LIN {X 0,Y 132.455,Z 460.625,A -85,B 0,C 180,E1 -25055.709,E2 -25055.709} C_VEL
LIN {X 0,Y 133.664,Z 463.302,A -85,B 0,C 180,E1 -25057.206,E2 -25057.206} C_VEL
LIN {X 0,Y 135.745,Z 466.18,A -85,B 0,C 180,E1 -25059.267,E2 -25059.267} C_VEL
LIN {X 0,Y 139.703,Z 473.299,A -85,B 0,C 180,E1 -25063.516,E2 -25063.516} C_VEL
LIN {X 0,Y 143.057,Z 480.754,A -85,B 0,C 180,E1 -25067.47,E2 -25067.47} C_VEL
LIN {X 0,Y 145.337,Z 487.251,A -85,B 0,C 180,E1 -25070.689,E2 -25070.689} C_VEL
LIN {X 0,Y 147.51,Z 495.449,A -85,B 0,C 180,E1 -25074.692,E2 -25074.692} C_VEL
LIN {X 0,Y 148.704,Z 503.562,A -85,B 0,C 180,E1 -25078.676,E2 -25078.676} C_VEL
LIN {X 0,Y 148.492,Z 505.004,A -85,B 0,C 180,E1 -25079.314,E2 -25079.314} C_VEL
LIN {X 0,Y 144.709,Z 513.242,A -85,B 0,C 180,E1 -25082.524,E2 -25082.524} C_VEL
LIN {X 0,Y 140.761,Z 521.094,A -85,B 0,C 180,E1 -25086.458,E2 -25086.458} C_VEL
LIN {X 0,Y 137.597,Z 527.354,A -85,B 0,C 180,E1 -25090.61,E2 -25090.61} C_VEL
LIN {X 0,Y 134.854,Z 532.346,A -85,B 0,C 180,E1 -25094.896,E2 -25094.896} C_VEL
LIN {X 0,Y 132.714,Z 536.229,A -85,B 0,C 180,E1 -25099.319,E2 -25099.319} C_VEL
LIN {X 0,Y 131.093,Z 539.121,A -85,B 0,C 180,E1 -25103.845,E2 -25103.845} C_VEL
LIN {X 0,Y 130.431,Z 540.5,A -85,B 0,C 180,E1 -25106.912,E2 -25106.912} C_VEL
LIN {X 0,Y 130.214,Z 542.071,A -85,B 0,C 180,E1 -25113.095,E2 -25113.095} C_VEL
LIN {X 0,Y 130.346,Z 542.325,A -85,B 0,C 180,E1 -25116.191,E2 -25116.191} C_VEL
LIN {X 0,Y 130.708,Z 542.169,A -85,B 0,C 180,E1 -25119.283,E2 -25119.283} C_VEL
LIN {X 0,Y 133.029,Z 540.615,A -85,B 0,C 180,E1 -25125.317,E2 -25125.317} C_VEL
LIN {X 0,Y 134.623,Z 539.262,A -85,B 0,C 180,E1 -25128.255,E2 -25128.255} C_VEL
LIN {X 0,Y 137.536,Z 536.056,A -85,B 0,C 180,E1 -25133.103,E2 -25133.103} C_VEL
LIN {X 0,Y 141.54,Z 531.107,A -85,B 0,C 180,E1 -25138.146,E2 -25138.146} C_VEL
LIN {X 0,Y 145.353,Z 525.767,A -85,B 0,C 180,E1 -25142.132,E2 -25142.132} C_VEL
LIN {X 0,Y 149.813,Z 519.05,A -85,B 0,C 180,E1 -25145.903,E2 -25145.903} C_VEL
LIN {X 0,Y 152.887,Z 513.993,A -85,B 0,C 180,E1 -25148.135,E2 -25148.135} C_VEL
LIN {X 0,Y 153.42,Z 512.528,A -85,B 0,C 180,E1 -25148.853,E2 -25148.853} C_VEL
LIN {X 0,Y 153.039,Z 506.128,A -85,B 0,C 180,E1 -25152.712,E2 -25152.712} C_VEL
LIN {X 0,Y 152.175,Z 500.29,A -85,B 0,C 180,E1 -25156.151,E2 -25156.151} C_VEL
LIN {X 0,Y 150.593,Z 493.774,A -85,B 0,C 180,E1 -25160.084,E2 -25160.084} C_VEL
LIN {X 0,Y 148.374,Z 487.095,A -85,B 0,C 180,E1 -25164.311,E2 -25164.311} C_VEL
LIN {X 0,Y 146.121,Z 481.755,A -85,B 0,C 180,E1 -25168.057,E2 -25168.057} C_VEL
LIN {X 0,Y 143.486,Z 476.383,A -85,B 0,C 180,E1 -25172.267,E2 -25172.267} C_VEL
LIN {X 0,Y 141.705,Z 473.457,A -85,B 0,C 180,E1 -25175.066,E2 -25175.066} C_VEL
LIN {X 0,Y 140.997,Z 471.644,A -85,B 0,C 180,E1 -25176.499,E2 -25176.499} C_VEL
LIN {X 0,Y 140.073,Z 470.683,A -85,B 0,C 180,E1 -25177.895,E2 -25177.895} C_VEL
LIN {X 0,Y 138.51,Z 471.715,A -85,B 0,C 180,E1 -25179.195,E2 -25179.195} C_VEL
LIN {X 0,Y 137.186,Z 472.293,A -85,B 0,C 180,E1 -25180.549,E2 -25180.549} C_VEL
LIN {X 0,Y 136.277,Z 473.332,A -85,B 0,C 180,E1 -25181.196,E2 -25181.196} C_VEL
LIN {X 0,Y 134.058,Z 476.489,A -85,B 0,C 180,E1 -25182.544,E2 -25182.544} C_VEL
LIN {X 0,Y 133.026,Z 477.829,A -85,B 0,C 180,E1 -25183.286,E2 -25183.286} C_VEL
LIN {X 0,Y 131.762,Z 479.038,A -85,B 0,C 180,E1 -25184.532,E2 -25184.532} C_VEL
LIN {X 0,Y 131.276,Z 479.221,A -85,B 0,C 180,E1 -25185.294,E2 -25185.294} C_VEL
LIN {X 0,Y 131.17,Z 478.619,A -85,B 0,C 180,E1 -25186.101,E2 -25186.101} C_VEL
LIN {X 0,Y 130.057,Z 490.324,A -85,B 0,C 180,E1 -25189.885,E2 -25189.885} C_VEL
LIN {X 0,Y 129.323,Z 500.383,A -85,B 0,C 180,E1 -25193.76,E2 -25193.76} C_VEL
LIN {X 0,Y 129.054,Z 510.666,A -85,B 0,C 180,E1 -25198.439,E2 -25198.439} C_VEL
LIN {X 0,Y 129.652,Z 520.617,A -85,B 0,C 180,E1 -25203.885,E2 -25203.885} C_VEL
LIN {X 0,Y 131.03,Z 528.937,A -85,B 0,C 180,E1 -25209.259,E2 -25209.259} C_VEL
LIN {X 0,Y 134.097,Z 536.791,A -85,B 0,C 180,E1 -25215.191,E2 -25215.191} C_VEL
LIN {X 0,Y 138.864,Z 543.178,A -85,B 0,C 180,E1 -25220.749,E2 -25220.749} C_VEL
LIN {X 0,Y 144.895,Z 548.225,A -85,B 0,C 180,E1 -25225.883,E2 -25225.883} C_VEL
LIN {X 0,Y 152.196,Z 551.996,A -85,B 0,C 180,E1 -25230.527,E2 -25230.527} C_VEL
LIN {X 0,Y 160.602,Z 554.573,A -85,B 0,C 180,E1 -25234.672,E2 -25234.672} C_VEL
LIN {X 0,Y 171.114,Z 556.077,A -85,B 0,C 180,E1 -25238.705,E2 -25238.705} C_VEL
LIN {X 0,Y 173.413,Z 556.275,A -85,B 0,C 180,E1 -25239.643,E2 -25239.643} C_VEL
LIN {X 0,Y 164.631,Z 559.404,A -85,B 0,C 180,E1 -25243.47,E2 -25243.47} C_VEL
LIN {X 0,Y 151.897,Z 562.596,A -85,B 0,C 180,E1 -25249.626,E2 -25249.626} C_VEL
LIN {X 0,Y 144.624,Z 563.745,A -85,B 0,C 180,E1 -25254.327,E2 -25254.327} C_VEL
LIN {X 0,Y 137.24,Z 563.903,A -85,B 0,C 180,E1 -25260.982,E2 -25260.982} C_VEL
LIN {X 0,Y 136.599,Z 564.145,A -85,B 0,C 180,E1 -25261.627,E2 -25261.627} C_VEL
LIN {X 0,Y 132.236,Z 569.84,A -85,B 0,C 180,E1 -25266.508,E2 -25266.508} C_VEL
LIN {X 0,Y 129.732,Z 573.62,A -85,B 0,C 180,E1 -25271.031,E2 -25271.031} C_VEL
LIN {X 0,Y 128.674,Z 575.62,A -85,B 0,C 180,E1 -25274.151,E2 -25274.151} C_VEL
LIN {X 0,Y 127.892,Z 578.343,A -85,B 0,C 180,E1 -25280.51,E2 -25280.51} C_VEL
LIN {X 0,Y 128.152,Z 579.135,A -85,B 0,C 180,E1 -25283.702,E2 -25283.702} C_VEL
LIN {X 0,Y 128.639,Z 579.512,A -85,B 0,C 180,E1 -25286.867,E2 -25286.867} C_VEL
LIN {X 0,Y 129.364,Z 579.441,A -85,B 0,C 180,E1 -25289.999,E2 -25289.999} C_VEL
LIN {X 0,Y 128.652,Z 578.72,A -85,B 0,C 180,E1 -25293.131,E2 -25293.131} C_VEL
LIN {X 0,Y 127.97,Z 576.442,A -85,B 0,C 180,E1 -25298.683,E2 -25298.683} C_VEL
LIN {X 0,Y 128.234,Z 572.826,A -85,B 0,C 180,E1 -25304.277,E2 -25304.277} C_VEL
LIN {X 0,Y 129.379,Z 568.573,A -85,B 0,C 180,E1 -25309.021,E2 -25309.021} C_VEL
LIN {X 0,Y 132.123,Z 562.165,A -85,B 0,C 180,E1 -25314.345,E2 -25314.345} C_VEL
LIN {X 0,Y 134.691,Z 556.486,A -85,B 0,C 180,E1 -25318.008,E2 -25318.008} C_VEL
LIN {X 0,Y 137.421,Z 547.961,A -85,B 0,C 180,E1 -25322.478,E2 -25322.478} C_VEL
LIN {X 0,Y 140.149,Z 538.592,A -85,B 0,C 180,E1 -25326.413,E2 -25326.413} C_VEL
LIN {X 0,Y 142.414,Z 528.505,A -85,B 0,C 180,E1 -25329.906,E2 -25329.906} C_VEL
LIN {X 0,Y 144.054,Z 517.734,A -85,B 0,C 180,E1 -25333.079,E2 -25333.079} C_VEL
LIN {X 0,Y 145.067,Z 506.101,A -85,B 0,C 180,E1 -25336.048,E2 -25336.048} C_VEL
LIN {X 0,Y 145.054,Z 495.817,A -85,B 0,C 180,E1 -25338.484,E2 -25338.484} C_VEL
LIN {X 0,Y 142.546,Z 488.232,A -85,B 0,C 180,E1 -25341.052,E2 -25341.052} C_VEL
LIN {X 0,Y 139.792,Z 481.393,A -85,B 0,C 180,E1 -25343.582,E2 -25343.582} C_VEL
LIN {X 0,Y 137.388,Z 475.79,A -85,B 0,C 180,E1 -25345.758,E2 -25345.758} C_VEL
LIN {X 0,Y 135.102,Z 471.173,A -85,B 0,C 180,E1 -25347.778,E2 -25347.778} C_VEL
LIN {X 0,Y 134.46,Z 469.699,A -85,B 0,C 180,E1 -25348.378,E2 -25348.378} C_VEL
LIN {X 0,Y 131.756,Z 465.595,A -85,B 0,C 180,E1 -25350.738,E2 -25350.738} C_VEL
LIN {X 0,Y 130.923,Z 463.575,A -85,B 0,C 180,E1 -25351.576,E2 -25351.576} C_VEL
LIN {X 0,Y 130.035,Z 462.484,A -85,B 0,C 180,E1 -25352.488,E2 -25352.488} C_VEL
LIN {X 0,Y 123.354,Z 459.002,A -85,B 0,C 180,E1 -25361.308,E2 -25361.308} C_VEL
LIN {X 0,Y 122.315,Z 457.065,A -85,B 0,C 180,E1 -25365.126,E2 -25365.126} C_VEL
LIN {X 0,Y 122.285,Z 456.255,A -85,B 0,C 180,E1 -25367.175,E2 -25367.175} C_VEL
LIN {X 0,Y 122.406,Z 456.239,A -85,B 0,C 180,E1 -25370.082,E2 -25370.082} C_VEL
LIN {X 0,Y 122.6,Z 456.214,A -85,B 0,C 180,E1 -25376.714,E2 -25376.714} C_VEL
LIN {X 0,Y 123.044,Z 456.158,A -85,B 0,C 180,E1 -25380.001,E2 -25380.001} C_VEL
LIN {X 0,Y 122.422,Z 456.217,A -85,B 0,C 180,E1 -25387.189,E2 -25387.189} C_VEL
LIN {X 0,Y 122.364,Z 456.225,A -85,B 0,C 180,E1 -25392.475,E2 -25392.475} C_VEL
LIN {X 0,Y 122.111,Z 456.272,A -85,B 0,C 180,E1 -25396.725,E2 -25396.725} C_VEL
LIN {X 0,Y 122.023,Z 456.226,A -85,B 0,C 180,E1 -25402.851,E2 -25402.851} C_VEL
LIN {X 0,Y 121.996,Z 456.337,A -85,B 0,C 180,E1 -25405.257,E2 -25405.257} C_VEL
LIN {X 0,Y 122.866,Z 458.968,A -85,B 0,C 180,E1 -25407.003,E2 -25407.003} C_VEL
LIN {X 0,Y 124.931,Z 461.19,A -85,B 0,C 180,E1 -25409.77,E2 -25409.77} C_VEL
LIN {X 0,Y 125.888,Z 461.888,A -85,B 0,C 180,E1 -25410.859,E2 -25410.859} C_VEL
LIN {X 0,Y 126.494,Z 463.534,A -85,B 0,C 180,E1 -25411.859,E2 -25411.859} C_VEL
LIN {X 0,Y 128.545,Z 466.286,A -85,B 0,C 180,E1 -25414.392,E2 -25414.392} C_VEL
LIN {X 0,Y 131.443,Z 470.995,A -85,B 0,C 180,E1 -25417.944,E2 -25417.944} C_VEL
LIN {X 0,Y 135.048,Z 478.23,A -85,B 0,C 180,E1 -25422.574,E2 -25422.574} C_VEL
LIN {X 0,Y 137.872,Z 484.993,A -85,B 0,C 180,E1 -25426.493,E2 -25426.493} C_VEL
LIN {X 0,Y 139.765,Z 490.991,A -85,B 0,C 180,E1 -25429.756,E2 -25429.756} C_VEL
LIN {X 0,Y 141.404,Z 497.843,A -85,B 0,C 180,E1 -25433.387,E2 -25433.387} C_VEL
LIN {X 0,Y 142.34,Z 504.865,A -85,B 0,C 180,E1 -25437.104,E2 -25437.104} C_VEL
LIN {X 0,Y 142.21,Z 506.847,A -85,B 0,C 180,E1 -25438.105,E2 -25438.105} C_VEL
LIN {X 0,Y 137.797,Z 515.869,A -85,B 0,C 180,E1 -25441.851,E2 -25441.851} C_VEL
LIN {X 0,Y 133.795,Z 523.357,A -85,B 0,C 180,E1 -25445.978,E2 -25445.978} C_VEL
LIN {X 0,Y 129.954,Z 530.239,A -85,B 0,C 180,E1 -25451.066,E2 -25451.066} C_VEL
LIN {X 0,Y 127.303,Z 534.822,A -85,B 0,C 180,E1 -25455.616,E2 -25455.616} C_VEL
LIN {X 0,Y 125.097,Z 538.361,A -85,B 0,C 180,E1 -25460.298,E2 -25460.298} C_VEL
LIN {X 0,Y 124.126,Z 540.175,A -85,B 0,C 180,E1 -25463.499,E2 -25463.499} C_VEL
LIN {X 0,Y 123.141,Z 542.507,A -85,B 0,C 180,E1 -25470.001,E2 -25470.001} C_VEL
LIN {X 0,Y 123.196,Z 543.097,A -85,B 0,C 180,E1 -25473.271,E2 -25473.271} C_VEL
LIN {X 0,Y 123.358,Z 543.338,A -85,B 0,C 180,E1 -25476.543,E2 -25476.543} C_VEL
LIN {X 0,Y 123.771,Z 543.169,A -85,B 0,C 180,E1 -25479.809,E2 -25479.809} C_VEL
LIN {X 0,Y 126.263,Z 541.596,A -85,B 0,C 180,E1 -25486.16,E2 -25486.16} C_VEL
LIN {X 0,Y 127.965,Z 540.229,A -85,B 0,C 180,E1 -25489.241,E2 -25489.241} C_VEL
LIN {X 0,Y 131.106,Z 536.994,A -85,B 0,C 180,E1 -25494.314,E2 -25494.314} C_VEL
LIN {X 0,Y 135.359,Z 532.034,A -85,B 0,C 180,E1 -25499.555,E2 -25499.555} C_VEL
LIN {X 0,Y 139.441,Z 526.67,A -85,B 0,C 180,E1 -25503.671,E2 -25503.671} C_VEL
LIN {X 0,Y 144.166,Z 519.925,A -85,B 0,C 180,E1 -25507.545,E2 -25507.545} C_VEL
LIN {X 0,Y 146.804,Z 515.846,A -85,B 0,C 180,E1 -25509.409,E2 -25509.409} C_VEL
LIN {X 0,Y 147.217,Z 514.42,A -85,B 0,C 180,E1 -25510.196,E2 -25510.196} C_VEL
LIN {X 0,Y 146.998,Z 508.333,A -85,B 0,C 180,E1 -25514.179,E2 -25514.179} C_VEL
LIN {X 0,Y 146.079,Z 501.501,A -85,B 0,C 180,E1 -25518.584,E2 -25518.584} C_VEL
LIN {X 0,Y 144.382,Z 494.701,A -85,B 0,C 180,E1 -25523.183,E2 -25523.183} C_VEL
LIN {X 0,Y 142.625,Z 489.08,A -85,B 0,C 180,E1 -25527.177,E2 -25527.177} C_VEL
LIN {X 0,Y 141.15,Z 485.34,A -85,B 0,C 180,E1 -25530.137,E2 -25530.137} C_VEL
LIN {X 0,Y 138.841,Z 480.634,A -85,B 0,C 180,E1 -25534.515,E2 -25534.515} C_VEL
LIN {X 0,Y 137.906,Z 478.488,A -85,B 0,C 180,E1 -25536.539,E2 -25536.539} C_VEL
LIN {X 0,Y 135.982,Z 478.364,A -85,B 0,C 180,E1 -25538.79,E2 -25538.79} C_VEL
LIN {X 0,Y 135.185,Z 479.091,A -85,B 0,C 180,E1 -25539.358,E2 -25539.358} C_VEL
LIN {X 0,Y 131.792,Z 483.155,A -85,B 0,C 180,E1 -25541.339,E2 -25541.339} C_VEL
LIN {X 0,Y 130.15,Z 484.651,A -85,B 0,C 180,E1 -25542.722,E2 -25542.722} C_VEL
LIN {X 0,Y 128.889,Z 485.514,A -85,B 0,C 180,E1 -25544.178,E2 -25544.178} C_VEL
LIN {X 0,Y 128.124,Z 486.286,A -85,B 0,C 180,E1 -25544.902,E2 -25544.902} C_VEL
LIN {X 0,Y 125.203,Z 490.091,A -85,B 0,C 180,E1 -25547.024,E2 -25547.024} C_VEL
LIN {X 0,Y 123.779,Z 491.683,A -85,B 0,C 180,E1 -25548.537,E2 -25548.537} C_VEL
LIN {X 0,Y 122.92,Z 492.401,A -85,B 0,C 180,E1 -25550.123,E2 -25550.123} C_VEL
LIN {X 0,Y 122.915,Z 491.967,A -85,B 0,C 180,E1 -25551.16,E2 -25551.16} C_VEL
LIN {X 0,Y 122.168,Z 503.178,A -85,B 0,C 180,E1 -25555.876,E2 -25555.876} C_VEL
LIN {X 0,Y 122.357,Z 514.588,A -85,B 0,C 180,E1 -25561.645,E2 -25561.645} C_VEL
LIN {X 0,Y 123.198,Z 522.776,A -85,B 0,C 180,E1 -25566.551,E2 -25566.551} C_VEL
LIN {X 0,Y 125.498,Z 531.937,A -85,B 0,C 180,E1 -25572.944,E2 -25572.944} C_VEL
LIN {X 0,Y 129.54,Z 539.473,A -85,B 0,C 180,E1 -25578.997,E2 -25578.997} C_VEL
LIN {X 0,Y 135.24,Z 545.612,A -85,B 0,C 180,E1 -25584.565,E2 -25584.565} C_VEL
LIN {X 0,Y 142.224,Z 550.434,A -85,B 0,C 180,E1 -25589.613,E2 -25589.613} C_VEL
LIN {X 0,Y 150.409,Z 554.051,A -85,B 0,C 180,E1 -25594.105,E2 -25594.105} C_VEL
LIN {X 0,Y 159.616,Z 556.514,A -85,B 0,C 180,E1 -25598.055,E2 -25598.055} C_VEL
LIN {X 0,Y 163.325,Z 557.125,A -85,B 0,C 180,E1 -25599.398,E2 -25599.398} C_VEL
LIN {X 0,Y 162.612,Z 557.733,A -85,B 0,C 180,E1 -25600.413,E2 -25600.413} C_VEL
LIN {X 0,Y 150.789,Z 560.452,A -85,B 0,C 180,E1 -25605.642,E2 -25605.642} C_VEL
LIN {X 0,Y 142.696,Z 561.665,A -85,B 0,C 180,E1 -25610.187,E2 -25610.187} C_VEL
LIN {X 0,Y 135.717,Z 562.042,A -85,B 0,C 180,E1 -25615.275,E2 -25615.275} C_VEL
LIN {X 0,Y 131.687,Z 561.807,A -85,B 0,C 180,E1 -25619.118,E2 -25619.118} C_VEL
LIN {X 0,Y 126.903,Z 567.402,A -85,B 0,C 180,E1 -25623.701,E2 -25623.701} C_VEL
LIN {X 0,Y 123.803,Z 571.506,A -85,B 0,C 180,E1 -25628.346,E2 -25628.346} C_VEL
LIN {X 0,Y 121.805,Z 574.628,A -85,B 0,C 180,E1 -25633.231,E2 -25633.231} C_VEL
LIN {X 0,Y 120.852,Z 577.335,A -85,B 0,C 180,E1 -25639.952,E2 -25639.952} C_VEL
LIN {X 0,Y 121.06,Z 578.12,A -85,B 0,C 180,E1 -25643.332,E2 -25643.332} C_VEL
LIN {X 0,Y 121.547,Z 578.487,A -85,B 0,C 180,E1 -25646.685,E2 -25646.685} C_VEL
LIN {X 0,Y 122.269,Z 578.407,A -85,B 0,C 180,E1 -25649.999,E2 -25649.999} C_VEL
LIN {X 0,Y 121.558,Z 577.676,A -85,B 0,C 180,E1 -25653.314,E2 -25653.314} C_VEL
LIN {X 0,Y 120.913,Z 575.542,A -85,B 0,C 180,E1 -25658.845,E2 -25658.845} C_VEL
LIN {X 0,Y 121.263,Z 571.729,A -85,B 0,C 180,E1 -25665.117,E2 -25665.117} C_VEL
LIN {X 0,Y 122.619,Z 567.463,A -85,B 0,C 180,E1 -25670.114,E2 -25670.114} C_VEL
LIN {X 0,Y 125.644,Z 561.032,A -85,B 0,C 180,E1 -25675.689,E2 -25675.689} C_VEL
LIN {X 0,Y 128.249,Z 555.298,A -85,B 0,C 180,E1 -25679.55,E2 -25679.55} C_VEL
LIN {X 0,Y 130.723,Z 548.31,A -85,B 0,C 180,E1 -25683.439,E2 -25683.439} C_VEL
LIN {X 0,Y 133.241,Z 540.477,A -85,B 0,C 180,E1 -25687.034,E2 -25687.034} C_VEL
LIN {X 0,Y 135.841,Z 530.634,A -85,B 0,C 180,E1 -25690.781,E2 -25690.781} C_VEL
LIN {X 0,Y 137.901,Z 519.873,A -85,B 0,C 180,E1 -25694.253,E2 -25694.253} C_VEL
LIN {X 0,Y 139.291,Z 508.603,A -85,B 0,C 180,E1 -25697.395,E2 -25697.395} C_VEL
LIN {X 0,Y 139.703,Z 499.821,A -85,B 0,C 180,E1 -25699.632,E2 -25699.632} C_VEL
LIN {X 0,Y 138.318,Z 494.611,A -85,B 0,C 180,E1 -25701.507,E2 -25701.507} C_VEL
LIN {X 0,Y 135.885,Z 487.069,A -85,B 0,C 180,E1 -25704.389,E2 -25704.389} C_VEL
LIN {X 0,Y 133.821,Z 481.653,A -85,B 0,C 180,E1 -25706.647,E2 -25706.647} C_VEL
LIN {X 0,Y 131.459,Z 476.49,A -85,B 0,C 180,E1 -25709.109,E2 -25709.109} C_VEL
LIN {X 0,Y 130.664,Z 474.81,A -85,B 0,C 180,E1 -25709.94,E2 -25709.94} C_VEL
LIN {X 0,Y 128.127,Z 470.019,A -85,B 0,C 180,E1 -25712.653,E2 -25712.653} C_VEL
LIN {X 0,Y 127.351,Z 468.142,A -85,B 0,C 180,E1 -25713.581,E2 -25713.581} C_VEL
LIN {X 0,Y 124.321,Z 463.748,A -85,B 0,C 180,E1 -25717.02,E2 -25717.02} C_VEL
LIN {X 0,Y 122.927,Z 460.205,A -85,B 0,C 180,E1 -25719.064,E2 -25719.064} C_VEL
LIN {X 0,Y 122.315,Z 457.065,A -85,B 0,C 180,E1 -25725.126,E2 -25725.126} C_VEL
LIN {X 0,Y 121.661,Z 456.408,A -85,B 0,C 180,E1 -25727.844,E2 -25727.844} C_VEL
LIN {X 0,Y 120.391,Z 456.491,A -85,B 0,C 180,E1 -25730.582,E2 -25730.582} C_VEL
LIN {X 0,Y 115.974,Z 457.038,A -85,B 0,C 180,E1 -25740.108,E2 -25740.108} C_VEL
LIN {X 0,Y 115.388,Z 457.094,A -85,B 0,C 180,E1 -25747.09,E2 -25747.09} C_VEL
LIN {X 0,Y 115.285,Z 457.106,A -85,B 0,C 180,E1 -25752.74,E2 -25752.74} C_VEL
LIN {X 0,Y 115.157,Z 457.253,A -85,B 0,C 180,E1 -25754.469,E2 -25754.469} C_VEL
LIN {X 0,Y 115.627,Z 459.156,A -85,B 0,C 180,E1 -25756.554,E2 -25756.554} C_VEL
LIN {X 0,Y 117.482,Z 461.685,A -85,B 0,C 180,E1 -25761.035,E2 -25761.035} C_VEL
LIN {X 0,Y 119.357,Z 462.892,A -85,B 0,C 180,E1 -25764.223,E2 -25764.223} C_VEL
LIN {X 0,Y 120.117,Z 465.17,A -85,B 0,C 180,E1 -25766.029,E2 -25766.029} C_VEL
LIN {X 0,Y 122.189,Z 467.655,A -85,B 0,C 180,E1 -25769.269,E2 -25769.269} C_VEL
LIN {X 0,Y 125.361,Z 472.867,A -85,B 0,C 180,E1 -25774.099,E2 -25774.099} C_VEL
LIN {X 0,Y 128.07,Z 478.065,A -85,B 0,C 180,E1 -25778.124,E2 -25778.124} C_VEL
LIN {X 0,Y 131.219,Z 485.328,A -85,B 0,C 180,E1 -25783.069,E2 -25783.069} C_VEL
LIN {X 0,Y 133.616,Z 492.365,A -85,B 0,C 180,E1 -25787.425,E2 -25787.425} C_VEL
LIN {X 0,Y 135.158,Z 499.241,A -85,B 0,C 180,E1 -25791.393,E2 -25791.393} C_VEL
LIN {X 0,Y 136.083,Z 506.163,A -85,B 0,C 180,E1 -25795.383,E2 -25795.383} C_VEL
LIN {X 0,Y 135.981,Z 508.704,A -85,B 0,C 180,E1 -25796.785,E2 -25796.785} C_VEL
LIN {X 0,Y 131.656,Z 517.036,A -85,B 0,C 180,E1 -25800.411,E2 -25800.411} C_VEL
LIN {X 0,Y 127.428,Z 524.488,A -85,B 0,C 180,E1 -25804.696,E2 -25804.696} C_VEL
LIN {X 0,Y 123.34,Z 531.349,A -85,B 0,C 180,E1 -25810.009,E2 -25810.009} C_VEL
LIN {X 0,Y 120.522,Z 535.91,A -85,B 0,C 180,E1 -25814.788,E2 -25814.788} C_VEL
LIN {X 0,Y 118.194,Z 539.429,A -85,B 0,C 180,E1 -25819.725,E2 -25819.725} C_VEL
LIN {X 0,Y 117.161,Z 541.227,A -85,B 0,C 180,E1 -25823.11,E2 -25823.11} C_VEL
LIN {X 0,Y 116.114,Z 543.541,A -85,B 0,C 180,E1 -25830.001,E2 -25830.001} C_VEL
LIN {X 0,Y 116.179,Z 544.122,A -85,B 0,C 180,E1 -25833.469,E2 -25833.469} C_VEL
LIN {X 0,Y 116.376,Z 544.349,A -85,B 0,C 180,E1 -25836.938,E2 -25836.938} C_VEL
LIN {X 0,Y 116.846,Z 544.168,A -85,B 0,C 180,E1 -25840.396,E2 -25840.396} C_VEL
LIN {X 0,Y 119.527,Z 542.578,A -85,B 0,C 180,E1 -25847.098,E2 -25847.098} C_VEL
LIN {X 0,Y 121.348,Z 541.195,A -85,B 0,C 180,E1 -25850.335,E2 -25850.335} C_VEL
LIN {X 0,Y 124.675,Z 537.987,A -85,B 0,C 180,E1 -25855.585,E2 -25855.585} C_VEL
LIN {X 0,Y 129.276,Z 532.96,A -85,B 0,C 180,E1 -25861.096,E2 -25861.096} C_VEL
LIN {X 0,Y 133.639,Z 527.573,A -85,B 0,C 180,E1 -25865.345,E2 -25865.345} C_VEL
LIN {X 0,Y 138.648,Z 520.797,A -85,B 0,C 180,E1 -25869.319,E2 -25869.319} C_VEL
LIN {X 0,Y 140.429,Z 518.156,A -85,B 0,C 180,E1 -25870.588,E2 -25870.588} C_VEL
LIN {X 0,Y 141.059,Z 516.368,A -85,B 0,C 180,E1 -25871.638,E2 -25871.638} C_VEL
LIN {X 0,Y 141.062,Z 510.539,A -85,B 0,C 180,E1 -25875.771,E2 -25875.771} C_VEL
LIN {X 0,Y 140.311,Z 504.146,A -85,B 0,C 180,E1 -25880.336,E2 -25880.336} C_VEL
LIN {X 0,Y 138.884,Z 497.463,A -85,B 0,C 180,E1 -25885.298,E2 -25885.298} C_VEL
LIN {X 0,Y 137.447,Z 492.606,A -85,B 0,C 180,E1 -25889.247,E2 -25889.247} C_VEL
LIN {X 0,Y 136.197,Z 489.227,A -85,B 0,C 180,E1 -25892.327,E2 -25892.327} C_VEL
LIN {X 0,Y 134.942,Z 486.202,A -85,B 0,C 180,E1 -25895.376,E2 -25895.376} C_VEL
LIN {X 0,Y 134.329,Z 484.84,A -85,B 0,C 180,E1 -25896.896,E2 -25896.896} C_VEL
LIN {X 0,Y 132.468,Z 486.274,A -85,B 0,C 180,E1 -25898.199,E2 -25898.199} C_VEL
LIN {X 0,Y 130.201,Z 488.558,A -85,B 0,C 180,E1 -25899.46,E2 -25899.46} C_VEL
LIN {X 0,Y 128.393,Z 490.072,A -85,B 0,C 180,E1 -25900.826,E2 -25900.826} C_VEL
LIN {X 0,Y 126.092,Z 491.835,A -85,B 0,C 180,E1 -25902.985,E2 -25902.985} C_VEL
LIN {X 0,Y 123.137,Z 495.157,A -85,B 0,C 180,E1 -25904.948,E2 -25904.948} C_VEL
LIN {X 0,Y 121.358,Z 496.937,A -85,B 0,C 180,E1 -25906.605,E2 -25906.605} C_VEL
LIN {X 0,Y 119.394,Z 498.521,A -85,B 0,C 180,E1 -25909.828,E2 -25909.828} C_VEL
LIN {X 0,Y 117.692,Z 500.726,A -85,B 0,C 180,E1 -25911.414,E2 -25911.414} C_VEL
LIN {X 0,Y 116.319,Z 502.442,A -85,B 0,C 180,E1 -25913.059,E2 -25913.059} C_VEL
LIN {X 0,Y 115.043,Z 504.118,A -85,B 0,C 180,E1 -25916.497,E2 -25916.497} C_VEL
LIN {X 0,Y 115.224,Z 503.986,A -85,B 0,C 180,E1 -25917.378,E2 -25917.378} C_VEL
LIN {X 0,Y 115.562,Z 513.858,A -85,B 0,C 180,E1 -25922.614,E2 -25922.614} C_VEL
LIN {X 0,Y 116.745,Z 523.524,A -85,B 0,C 180,E1 -25928.655,E2 -25928.655} C_VEL
LIN {X 0,Y 119.587,Z 532.711,A -85,B 0,C 180,E1 -25935.334,E2 -25935.334} C_VEL
LIN {X 0,Y 124.295,Z 540.339,A -85,B 0,C 180,E1 -25941.563,E2 -25941.563} C_VEL
LIN {X 0,Y 130.525,Z 546.603,A -85,B 0,C 180,E1 -25947.237,E2 -25947.237} C_VEL
LIN {X 0,Y 138.115,Z 551.548,A -85,B 0,C 180,E1 -25952.296,E2 -25952.296} C_VEL
LIN {X 0,Y 149.206,Z 556.086,A -85,B 0,C 180,E1 -25957.758,E2 -25957.758} C_VEL
LIN {X 0,Y 154.137,Z 557.41,A -85,B 0,C 180,E1 -25959.668,E2 -25959.668} C_VEL
LIN {X 0,Y 150.425,Z 558.289,A -85,B 0,C 180,E1 -25961.622,E2 -25961.622} C_VEL
LIN {X 0,Y 137.435,Z 559.876,A -85,B 0,C 180,E1 -25968.333,E2 -25968.333} C_VEL
LIN {X 0,Y 128.064,Z 559.745,A -85,B 0,C 180,E1 -25975.404,E2 -25975.404} C_VEL
LIN {X 0,Y 126.675,Z 559.762,A -85,B 0,C 180,E1 -25976.704,E2 -25976.704} C_VEL
LIN {X 0,Y 121.999,Z 564.853,A -85,B 0,C 180,E1 -25980.681,E2 -25980.681} C_VEL
LIN {X 0,Y 118.2,Z 569.274,A -85,B 0,C 180,E1 -25985.404,E2 -25985.404} C_VEL
LIN {X 0,Y 116.325,Z 571.672,A -85,B 0,C 180,E1 -25988.745,E2 -25988.745} C_VEL
LIN {X 0,Y 114.98,Z 573.635,A -85,B 0,C 180,E1 -25992.204,E2 -25992.204} C_VEL
LIN {X 0,Y 113.813,Z 576.325,A -85,B 0,C 180,E1 -25999.323,E2 -25999.323} C_VEL
LIN {X 0,Y 113.955,Z 577.101,A -85,B 0,C 180,E1 -26002.914,E2 -26002.914} C_VEL
LIN {X 0,Y 114.456,Z 577.461,A -85,B 0,C 180,E1 -26006.479,E2 -26006.479} C_VEL
LIN {X 0,Y 115.172,Z 577.373,A -85,B 0,C 180,E1 -26009.999,E2 -26009.999} C_VEL
LIN {X 0,Y 114.444,Z 576.629,A -85,B 0,C 180,E1 -26013.52,E2 -26013.52} C_VEL
LIN {X 0,Y 113.847,Z 574.655,A -85,B 0,C 180,E1 -26018.992,E2 -26018.992} C_VEL
LIN {X 0,Y 114.074,Z 571.805,A -85,B 0,C 180,E1 -26024.266,E2 -26024.266} C_VEL
LIN {X 0,Y 115.264,Z 567.874,A -85,B 0,C 180,E1 -26029.593,E2 -26029.593} C_VEL
LIN {X 0,Y 117.597,Z 562.85,A -85,B 0,C 180,E1 -26034.729,E2 -26034.729} C_VEL
LIN {X 0,Y 121.022,Z 556.345,A -85,B 0,C 180,E1 -26039.765,E2 -26039.765} C_VEL
LIN {X 0,Y 124.064,Z 548.614,A -85,B 0,C 180,E1 -26044.505,E2 -26044.505} C_VEL
LIN {X 0,Y 127.137,Z 539.882,A -85,B 0,C 180,E1 -26048.775,E2 -26048.775} C_VEL
LIN {X 0,Y 130.159,Z 529.301,A -85,B 0,C 180,E1 -26052.975,E2 -26052.975} C_VEL
LIN {X 0,Y 132.477,Z 518.3,A -85,B 0,C 180,E1 -26056.65,E2 -26056.65} C_VEL
LIN {X 0,Y 133.846,Z 508.069,A -85,B 0,C 180,E1 -26059.654,E2 -26059.654} C_VEL
LIN {X 0,Y 134.253,Z 502.86,A -85,B 0,C 180,E1 -26061.084,E2 -26061.084} C_VEL
LIN {X 0,Y 133.142,Z 498.119,A -85,B 0,C 180,E1 -26062.957,E2 -26062.957} C_VEL
LIN {X 0,Y 130.611,Z 489.883,A -85,B 0,C 180,E1 -26066.528,E2 -26066.528} C_VEL
LIN {X 0,Y 129.063,Z 485.368,A -85,B 0,C 180,E1 -26068.6,E2 -26068.6} C_VEL
LIN {X 0,Y 127.001,Z 480.17,A -85,B 0,C 180,E1 -26071.266,E2 -26071.266} C_VEL
LIN {X 0,Y 124.723,Z 475.139,A -85,B 0,C 180,E1 -26074.24,E2 -26074.24} C_VEL
LIN {X 0,Y 124.141,Z 473.778,A -85,B 0,C 180,E1 -26075.039,E2 -26075.039} C_VEL
LIN {X 0,Y 121.517,Z 469.319,A -85,B 0,C 180,E1 -26078.588,E2 -26078.588} C_VEL
LIN {X 0,Y 120.353,Z 466.21,A -85,B 0,C 180,E1 -26080.603,E2 -26080.603} C_VEL
LIN {X 0,Y 115.633,Z 458.364,A -85,B 0,C 180,E1 -26090.048,E2 -26090.048} C_VEL
LIN {X 0,Y 115.336,Z 457.121,A -85,B 0,C 180,E1 -26091.238,E2 -26091.238} C_VEL
LIN {X 0,Y 115.974,Z 457.038,A -85,B 0,C 180,E1 -26100.108,E2 -26100.108} C_VEL
LIN {X 0,Y 115.297,Z 457.534,A -85,B 0,C 180,E1 -26103.011,E2 -26103.011} C_VEL
LIN {X 0,Y 114.014,Z 459.882,A -85,B 0,C 180,E1 -26107.773,E2 -26107.773} C_VEL
LIN {X 0,Y 113.446,Z 465.479,A -85,B 0,C 180,E1 -26115.347,E2 -26115.347} C_VEL
LIN {X 0,Y 114.124,Z 467.11,A -85,B 0,C 180,E1 -26117.934,E2 -26117.934} C_VEL
LIN {X 0,Y 116.457,Z 469.225,A -85,B 0,C 180,E1 -26123.096,E2 -26123.096} C_VEL
LIN {X 0,Y 117.062,Z 471.099,A -85,B 0,C 180,E1 -26124.851,E2 -26124.851} C_VEL
LIN {X 0,Y 118.818,Z 473.651,A -85,B 0,C 180,E1 -26128.243,E2 -26128.243} C_VEL
LIN {X 0,Y 122.026,Z 479.721,A -85,B 0,C 180,E1 -26134.163,E2 -26134.163} C_VEL
LIN {X 0,Y 123.831,Z 483.555,A -85,B 0,C 180,E1 -26137.386,E2 -26137.386} C_VEL
LIN {X 0,Y 126.704,Z 491.219,A -85,B 0,C 180,E1 -26143.006,E2 -26143.006} C_VEL
LIN {X 0,Y 128.439,Z 497.537,A -85,B 0,C 180,E1 -26147.221,E2 -26147.221} C_VEL
LIN {X 0,Y 129.542,Z 504.02,A -85,B 0,C 180,E1 -26151.304,E2 -26151.304} C_VEL
LIN {X 0,Y 129.927,Z 508.668,A -85,B 0,C 180,E1 -26154.232,E2 -26154.232} C_VEL
LIN {X 0,Y 129.821,Z 510.598,A -85,B 0,C 180,E1 -26155.364,E2 -26155.364} C_VEL
LIN {X 0,Y 124.807,Z 519.527,A -85,B 0,C 180,E1 -26159.55,E2 -26159.55} C_VEL
LIN {X 0,Y 120.471,Z 526.704,A -85,B 0,C 180,E1 -26164.054,E2 -26164.054} C_VEL
LIN {X 0,Y 116.773,Z 532.457,A -85,B 0,C 180,E1 -26168.832,E2 -26168.832} C_VEL
LIN {X 0,Y 113.768,Z 536.998,A -85,B 0,C 180,E1 -26173.861,E2 -26173.861} C_VEL
LIN {X 0,Y 111.302,Z 540.497,A -85,B 0,C 180,E1 -26179.081,E2 -26179.081} C_VEL
LIN {X 0,Y 110.201,Z 542.278,A -85,B 0,C 180,E1 -26182.673,E2 -26182.673} C_VEL
LIN {X 0,Y 109.086,Z 544.575,A -85,B 0,C 180,E1 -26190.001,E2 -26190.001} C_VEL
LIN {X 0,Y 109.163,Z 545.148,A -85,B 0,C 180,E1 -26193.692,E2 -26193.692} C_VEL
LIN {X 0,Y 109.399,Z 545.358,A -85,B 0,C 180,E1 -26197.383,E2 -26197.383} C_VEL
LIN {X 0,Y 109.935,Z 545.168,A -85,B 0,C 180,E1 -26201.058,E2 -26201.058} C_VEL
LIN {X 0,Y 112.827,Z 543.56,A -85,B 0,C 180,E1 -26208.148,E2 -26208.148} C_VEL
LIN {X 0,Y 114.78,Z 542.16,A -85,B 0,C 180,E1 -26211.555,E2 -26211.555} C_VEL
LIN {X 0,Y 118.32,Z 538.975,A -85,B 0,C 180,E1 -26217.003,E2 -26217.003} C_VEL
LIN {X 0,Y 123.298,Z 533.886,A -85,B 0,C 180,E1 -26222.787,E2 -26222.787} C_VEL
LIN {X 0,Y 127.964,Z 528.476,A -85,B 0,C 180,E1 -26227.168,E2 -26227.168} C_VEL
LIN {X 0,Y 133.273,Z 521.668,A -85,B 0,C 180,E1 -26231.238,E2 -26231.238} C_VEL
LIN {X 0,Y 134.886,Z 519.068,A -85,B 0,C 180,E1 -26232.637,E2 -26232.637} C_VEL
LIN {X 0,Y 135.139,Z 513.768,A -85,B 0,C 180,E1 -26236.727,E2 -26236.727} C_VEL
LIN {X 0,Y 134.745,Z 508.002,A -85,B 0,C 180,E1 -26241.252,E2 -26241.252} C_VEL
LIN {X 0,Y 133.9,Z 502.614,A -85,B 0,C 180,E1 -26245.651,E2 -26245.651} C_VEL
LIN {X 0,Y 132.855,Z 497.825,A -85,B 0,C 180,E1 -26249.832,E2 -26249.832} C_VEL
LIN {X 0,Y 131.393,Z 492.976,A -85,B 0,C 180,E1 -26254.664,E2 -26254.664} C_VEL
LIN {X 0,Y 131.009,Z 492.049,A -85,B 0,C 180,E1 -26255.781,E2 -26255.781} C_VEL
LIN {X 0,Y 130.21,Z 492.248,A -85,B 0,C 180,E1 -26256.575,E2 -26256.575} C_VEL
LIN {X 0,Y 128.479,Z 493.793,A -85,B 0,C 180,E1 -26257.485,E2 -26257.485} C_VEL
LIN {X 0,Y 126.506,Z 495.313,A -85,B 0,C 180,E1 -26258.831,E2 -26258.831} C_VEL
LIN {X 0,Y 124.827,Z 496.448,A -85,B 0,C 180,E1 -26260.256,E2 -26260.256} C_VEL
LIN {X 0,Y 120.58,Z 500.414,A -85,B 0,C 180,E1 -26263.056,E2 -26263.056} C_VEL
LIN {X 0,Y 118.819,Z 501.98,A -85,B 0,C 180,E1 -26264.563,E2 -26264.563} C_VEL
LIN {X 0,Y 116.422,Z 503.804,A -85,B 0,C 180,E1 -26267.802,E2 -26267.802} C_VEL
LIN {X 0,Y 113.284,Z 507.181,A -85,B 0,C 180,E1 -26270.897,E2 -26270.897} C_VEL
LIN {X 0,Y 112.134,Z 508.415,A -85,B 0,C 180,E1 -26272.798,E2 -26272.798} C_VEL
LIN {X 0,Y 110.882,Z 509.966,A -85,B 0,C 180,E1 -26276.365,E2 -26276.365} C_VEL
LIN {X 0,Y 109.684,Z 511.728,A -85,B 0,C 180,E1 -26278.163,E2 -26278.163} C_VEL
LIN {X 0,Y 108.872,Z 513.078,A -85,B 0,C 180,E1 -26279.999,E2 -26279.999} C_VEL
LIN {X 0,Y 108.812,Z 514.387,A -85,B 0,C 180,E1 -26284.166,E2 -26284.166} C_VEL
LIN {X 0,Y 108.993,Z 514.526,A -85,B 0,C 180,E1 -26284.623,E2 -26284.623} C_VEL
LIN {X 0,Y 110.502,Z 524.123,A -85,B 0,C 180,E1 -26290.999,E2 -26290.999} C_VEL
LIN {X 0,Y 113.89,Z 533.413,A -85,B 0,C 180,E1 -26297.971,E2 -26297.971} C_VEL
LIN {X 0,Y 119.243,Z 541.12,A -85,B 0,C 180,E1 -26304.366,E2 -26304.366} C_VEL
LIN {X 0,Y 126.079,Z 547.447,A -85,B 0,C 180,E1 -26310.111,E2 -26310.111} C_VEL
LIN {X 0,Y 134.305,Z 552.563,A -85,B 0,C 180,E1 -26315.142,E2 -26315.142} C_VEL
LIN {X 0,Y 143.664,Z 556.529,A -85,B 0,C 180,E1 -26319.491,E2 -26319.491} C_VEL
LIN {X 0,Y 143.852,Z 557.054,A -85,B 0,C 180,E1 -26320.425,E2 -26320.425} C_VEL
LIN {X 0,Y 132.38,Z 557.872,A -85,B 0,C 180,E1 -26326.356,E2 -26326.356} C_VEL
LIN {X 0,Y 122.137,Z 557.496,A -85,B 0,C 180,E1 -26333.954,E2 -26333.954} C_VEL
LIN {X 0,Y 115.877,Z 563.915,A -85,B 0,C 180,E1 -26338.966,E2 -26338.966} C_VEL
LIN {X 0,Y 111.776,Z 568.314,A -85,B 0,C 180,E1 -26343.887,E2 -26343.887} C_VEL
LIN {X 0,Y 109.705,Z 570.699,A -85,B 0,C 180,E1 -26347.394,E2 -26347.394} C_VEL
LIN {X 0,Y 108.206,Z 572.644,A -85,B 0,C 180,E1 -26351.049,E2 -26351.049} C_VEL
LIN {X 0,Y 106.795,Z 575.316,A -85,B 0,C 180,E1 -26358.613,E2 -26358.613} C_VEL
LIN {X 0,Y 106.861,Z 576.083,A -85,B 0,C 180,E1 -26362.441,E2 -26362.441} C_VEL
LIN {X 0,Y 107.363,Z 576.433,A -85,B 0,C 180,E1 -26366.246,E2 -26366.246} C_VEL
LIN {X 0,Y 108.071,Z 576.338,A -85,B 0,C 180,E1 -26369.999,E2 -26369.999} C_VEL
LIN {X 0,Y 107.317,Z 575.58,A -85,B 0,C 180,E1 -26373.754,E2 -26373.754} C_VEL
LIN {X 0,Y 106.779,Z 573.771,A -85,B 0,C 180,E1 -26379.151,E2 -26379.151} C_VEL
LIN {X 0,Y 107.107,Z 570.712,A -85,B 0,C 180,E1 -26385.216,E2 -26385.216} C_VEL
LIN {X 0,Y 108.535,Z 566.768,A -85,B 0,C 180,E1 -26390.863,E2 -26390.863} C_VEL
LIN {X 0,Y 111.147,Z 561.729,A -85,B 0,C 180,E1 -26396.27,E2 -26396.27} C_VEL
LIN {X 0,Y 114.523,Z 555.643,A -85,B 0,C 180,E1 -26401.235,E2 -26401.235} C_VEL
LIN {X 0,Y 117.426,Z 548.838,A -85,B 0,C 180,E1 -26405.699,E2 -26405.699} C_VEL
LIN {X 0,Y 120.895,Z 539.921,A -85,B 0,C 180,E1 -26410.387,E2 -26410.387} C_VEL
LIN {X 0,Y 124.026,Z 530.237,A -85,B 0,C 180,E1 -26414.526,E2 -26414.526} C_VEL
LIN {X 0,Y 126.743,Z 518.962,A -85,B 0,C 180,E1 -26418.557,E2 -26418.557} C_VEL
LIN {X 0,Y 128.488,Z 508.25,A -85,B 0,C 180,E1 -26421.912,E2 -26421.912} C_VEL
LIN {X 0,Y 128.784,Z 506.033,A -85,B 0,C 180,E1 -26422.564,E2 -26422.564} C_VEL
LIN {X 0,Y 128.23,Z 502.84,A -85,B 0,C 180,E1 -26423.902,E2 -26423.902} C_VEL
LIN {X 0,Y 125.98,Z 494.132,A -85,B 0,C 180,E1 -26427.997,E2 -26427.997} C_VEL
LIN {X 0,Y 124.507,Z 489.427,A -85,B 0,C 180,E1 -26430.403,E2 -26430.403} C_VEL
LIN {X 0,Y 123.014,Z 485.142,A -85,B 0,C 180,E1 -26432.803,E2 -26432.803} C_VEL
LIN {X 0,Y 120.727,Z 479.316,A -85,B 0,C 180,E1 -26436.522,E2 -26436.522} C_VEL
LIN {X 0,Y 118.367,Z 474.399,A -85,B 0,C 180,E1 -26440.49,E2 -26440.49} C_VEL
LIN {X 0,Y 117.588,Z 472.163,A -85,B 0,C 180,E1 -26442.163,E2 -26442.163} C_VEL
LIN {X 0,Y 113.808,Z 464.532,A -85,B 0,C 180,E1 -26451.566,E2 -26451.566} C_VEL
LIN {X 0,Y 113.716,Z 464.123,A -85,B 0,C 180,E1 -26452.006,E2 -26452.006} C_VEL
LIN {X 0,Y 111.967,Z 462.875,A -85,B 0,C 180,E1 -26460.001,E2 -26460.001} C_VEL
LIN {X 0,Y 113.16,Z 463.912,A -85,B 0,C 180,E1 -26473.333,E2 -26473.333} C_VEL
LIN {X 0,Y 113.446,Z 465.479,A -85,B 0,C 180,E1 -26475.347,E2 -26475.347} C_VEL
LIN {X 0,Y 114.061,Z 468.894,A -85,B 0,C 180,E1 -26478.93,E2 -26478.93} C_VEL
LIN {X 0,Y 115.127,Z 477.33,A -85,B 0,C 180,E1 -26485.661,E2 -26485.661} C_VEL
LIN {X 0,Y 116.106,Z 481.122,A -85,B 0,C 180,E1 -26489.097,E2 -26489.097} C_VEL
LIN {X 0,Y 118.402,Z 486.283,A -85,B 0,C 180,E1 -26494.324,E2 -26494.324} C_VEL
LIN {X 0,Y 120.232,Z 491.448,A -85,B 0,C 180,E1 -26498.709,E2 -26498.709} C_VEL
LIN {X 0,Y 121.698,Z 496.084,A -85,B 0,C 180,E1 -26502.363,E2 -26502.363} C_VEL
LIN {X 0,Y 122.988,Z 502.096,A -85,B 0,C 180,E1 -26506.708,E2 -26506.708} C_VEL
LIN {X 0,Y 123.749,Z 508.802,A -85,B 0,C 180,E1 -26511.339,E2 -26511.339} C_VEL
LIN {X 0,Y 123.72,Z 512.472,A -85,B 0,C 180,E1 -26513.816,E2 -26513.816} C_VEL
LIN {X 0,Y 118.82,Z 520.683,A -85,B 0,C 180,E1 -26517.837,E2 -26517.837} C_VEL
LIN {X 0,Y 114.211,Z 527.835,A -85,B 0,C 180,E1 -26522.516,E2 -26522.516} C_VEL
LIN {X 0,Y 110.262,Z 533.565,A -85,B 0,C 180,E1 -26527.516,E2 -26527.516} C_VEL
LIN {X 0,Y 107.048,Z 538.086,A -85,B 0,C 180,E1 -26532.817,E2 -26532.817} C_VEL
LIN {X 0,Y 104.424,Z 541.565,A -85,B 0,C 180,E1 -26538.352,E2 -26538.352} C_VEL
LIN {X 0,Y 103.247,Z 543.328,A -85,B 0,C 180,E1 -26542.176,E2 -26542.176} C_VEL
LIN {X 0,Y 102.381,Z 544.669,A -85,B 0,C 180,E1 -26546.065,E2 -26546.065} C_VEL
LIN {X 0,Y 102.149,Z 546.173,A -85,B 0,C 180,E1 -26553.946,E2 -26553.946} C_VEL
LIN {X 0,Y 102.43,Z 546.366,A -85,B 0,C 180,E1 -26557.888,E2 -26557.888} C_VEL
LIN {X 0,Y 103.041,Z 546.168,A -85,B 0,C 180,E1 -26561.808,E2 -26561.808} C_VEL
LIN {X 0,Y 106.17,Z 544.541,A -85,B 0,C 180,E1 -26569.329,E2 -26569.329} C_VEL
LIN {X 0,Y 108.27,Z 543.124,A -85,B 0,C 180,E1 -26572.923,E2 -26572.923} C_VEL
LIN {X 0,Y 112.069,Z 539.945,A -85,B 0,C 180,E1 -26578.602,E2 -26578.602} C_VEL
LIN {X 0,Y 117.44,Z 534.812,A -85,B 0,C 180,E1 -26584.648,E2 -26584.648} C_VEL
LIN {X 0,Y 122.431,Z 529.38,A -85,B 0,C 180,E1 -26589.158,E2 -26589.158} C_VEL
LIN {X 0,Y 127.849,Z 522.81,A -85,B 0,C 180,E1 -26593.177,E2 -26593.177} C_VEL
LIN {X 0,Y 128.761,Z 521.506,A -85,B 0,C 180,E1 -26593.871,E2 -26593.871} C_VEL
LIN {X 0,Y 129.238,Z 516.92,A -85,B 0,C 180,E1 -26597.785,E2 -26597.785} C_VEL
LIN {X 0,Y 129.163,Z 511.809,A -85,B 0,C 180,E1 -26602.175,E2 -26602.175} C_VEL
LIN {X 0,Y 128.668,Z 506.582,A -85,B 0,C 180,E1 -26606.892,E2 -26606.892} C_VEL
LIN {X 0,Y 127.841,Z 501.746,A -85,B 0,C 180,E1 -26611.595,E2 -26611.595} C_VEL
LIN {X 0,Y 127.363,Z 499.772,A -85,B 0,C 180,E1 -26613.803,E2 -26613.803} C_VEL
LIN {X 0,Y 126.068,Z 499.257,A -85,B 0,C 180,E1 -26615.757,E2 -26615.757} C_VEL
LIN {X 0,Y 122.645,Z 501.542,A -85,B 0,C 180,E1 -26618.131,E2 -26618.131} C_VEL
LIN {X 0,Y 118.111,Z 505.275,A -85,B 0,C 180,E1 -26620.894,E2 -26620.894} C_VEL
LIN {X 0,Y 116.16,Z 506.845,A -85,B 0,C 180,E1 -26622.391,E2 -26622.391} C_VEL
LIN {X 0,Y 113.299,Z 508.862,A -85,B 0,C 180,E1 -26625.633,E2 -26625.633} C_VEL
LIN {X 0,Y 109.823,Z 512.057,A -85,B 0,C 180,E1 -26628.931,E2 -26628.931} C_VEL
LIN {X 0,Y 107.668,Z 514.102,A -85,B 0,C 180,E1 -26632.498,E2 -26632.498} C_VEL
LIN {X 0,Y 106.949,Z 514.883,A -85,B 0,C 180,E1 -26634.343,E2 -26634.343} C_VEL
LIN {X 0,Y 104.753,Z 517.671,A -85,B 0,C 180,E1 -26638.075,E2 -26638.075} C_VEL
LIN {X 0,Y 104.224,Z 518.599,A -85,B 0,C 180,E1 -26639.999,E2 -26639.999} C_VEL
LIN {X 0,Y 104.057,Z 519.857,A -85,B 0,C 180,E1 -26643.872,E2 -26643.872} C_VEL
LIN {X 0,Y 103.071,Z 522.57,A -85,B 0,C 180,E1 -26647.837,E2 -26647.837} C_VEL
LIN {X 0,Y 103.554,Z 524.179,A -85,B 0,C 180,E1 -26651.747,E2 -26651.747} C_VEL
LIN {X 0,Y 104.413,Z 524.515,A -85,B 0,C 180,E1 -26653.502,E2 -26653.502} C_VEL
LIN {X 0,Y 109.156,Z 535.035,A -85,B 0,C 180,E1 -26661.728,E2 -26661.728} C_VEL
LIN {X 0,Y 116.29,Z 543.513,A -85,B 0,C 180,E1 -26668.912,E2 -26668.912} C_VEL
LIN {X 0,Y 124.169,Z 549.683,A -85,B 0,C 180,E1 -26674.472,E2 -26674.472} C_VEL
LIN {X 0,Y 133.309,Z 554.667,A -85,B 0,C 180,E1 -26679.244,E2 -26679.244} C_VEL
LIN {X 0,Y 134.45,Z 555.149,A -85,B 0,C 180,E1 -26679.741,E2 -26679.741} C_VEL
LIN {X 0,Y 133.544,Z 555.605,A -85,B 0,C 180,E1 -26680.98,E2 -26680.98} C_VEL
LIN {X 0,Y 123.385,Z 555.483,A -85,B 0,C 180,E1 -26686.879,E2 -26686.879} C_VEL
LIN {X 0,Y 118.02,Z 555.071,A -85,B 0,C 180,E1 -26690.96,E2 -26690.96} C_VEL
LIN {X 0,Y 111.661,Z 561.311,A -85,B 0,C 180,E1 -26695.495,E2 -26695.495} C_VEL
LIN {X 0,Y 106.779,Z 566.036,A -85,B 0,C 180,E1 -26700.419,E2 -26700.419} C_VEL
LIN {X 0,Y 103.158,Z 569.727,A -85,B 0,C 180,E1 -26705.871,E2 -26705.871} C_VEL
LIN {X 0,Y 101.491,Z 571.655,A -85,B 0,C 180,E1 -26709.742,E2 -26709.742} C_VEL
LIN {X 0,Y 99.798,Z 574.307,A -85,B 0,C 180,E1 -26717.802,E2 -26717.802} C_VEL
LIN {X 0,Y 99.783,Z 575.066,A -85,B 0,C 180,E1 -26721.901,E2 -26721.901} C_VEL
LIN {X 0,Y 100.269,Z 575.405,A -85,B 0,C 180,E1 -26725.98,E2 -26725.98} C_VEL
LIN {X 0,Y 100.964,Z 575.302,A -85,B 0,C 180,E1 -26729.999,E2 -26729.999} C_VEL
LIN {X 0,Y 100.196,Z 574.532,A -85,B 0,C 180,E1 -26734.021,E2 -26734.021} C_VEL
LIN {X 0,Y 99.722,Z 572.874,A -85,B 0,C 180,E1 -26739.37,E2 -26739.37} C_VEL
LIN {X 0,Y 100.197,Z 569.624,A -85,B 0,C 180,E1 -26746.293,E2 -26746.293} C_VEL
LIN {X 0,Y 101.878,Z 565.664,A -85,B 0,C 180,E1 -26752.297,E2 -26752.297} C_VEL
LIN {X 0,Y 104.789,Z 560.607,A -85,B 0,C 180,E1 -26757.999,E2 -26757.999} C_VEL
LIN {X 0,Y 107.36,Z 556.473,A -85,B 0,C 180,E1 -26761.68,E2 -26761.68} C_VEL
LIN {X 0,Y 110.853,Z 549.062,A -85,B 0,C 180,E1 -26767.033,E2 -26767.033} C_VEL
LIN {X 0,Y 114.183,Z 541.405,A -85,B 0,C 180,E1 -26771.426,E2 -26771.426} C_VEL
LIN {X 0,Y 117.617,Z 532.064,A -85,B 0,C 180,E1 -26775.81,E2 -26775.81} C_VEL
LIN {X 0,Y 120.763,Z 521.374,A -85,B 0,C 180,E1 -26779.987,E2 -26779.987} C_VEL
LIN {X 0,Y 123.059,Z 510.286,A -85,B 0,C 180,E1 -26783.772,E2 -26783.772} C_VEL
LIN {X 0,Y 123.318,Z 508.741,A -85,B 0,C 180,E1 -26784.257,E2 -26784.257} C_VEL
LIN {X 0,Y 121.658,Z 499.804,A -85,B 0,C 180,E1 -26788.674,E2 -26788.674} C_VEL
LIN {X 0,Y 119.672,Z 492.256,A -85,B 0,C 180,E1 -26792.927,E2 -26792.927} C_VEL
LIN {X 0,Y 117.614,Z 485.787,A -85,B 0,C 180,E1 -26797.145,E2 -26797.145} C_VEL
LIN {X 0,Y 115.492,Z 480.784,A -85,B 0,C 180,E1 -26801.369,E2 -26801.369} C_VEL
LIN {X 0,Y 114.393,Z 477.65,A -85,B 0,C 180,E1 -26804.18,E2 -26804.18} C_VEL
LIN {X 0,Y 111.73,Z 470.913,A -85,B 0,C 180,E1 -26812.773,E2 -26812.773} C_VEL
LIN {X 0,Y 110.212,Z 469.783,A -85,B 0,C 180,E1 -26820.001,E2 -26820.001} C_VEL
LIN {X 0,Y 110.597,Z 470.444,A -85,B 0,C 180,E1 -26830.991,E2 -26830.991} C_VEL
LIN {X 0,Y 112.863,Z 475.129,A -85,B 0,C 180,E1 -26840.926,E2 -26840.926} C_VEL
LIN {X 0,Y 113.286,Z 475.435,A -85,B 0,C 180,E1 -26841.854,E2 -26841.854} C_VEL
LIN {X 0,Y 116.106,Z 481.122,A -85,B 0,C 180,E1 -26849.097,E2 -26849.097} C_VEL
LIN {X 0,Y 116.813,Z 484.133,A -85,B 0,C 180,E1 -26851.581,E2 -26851.581} C_VEL
LIN {X 0,Y 116.939,Z 487.851,A -85,B 0,C 180,E1 -26853.86,E2 -26853.86} C_VEL
LIN {X 0,Y 116.295,Z 498.354,A -85,B 0,C 180,E1 -26859.84,E2 -26859.84} C_VEL
LIN {X 0,Y 116.515,Z 500.558,A -85,B 0,C 180,E1 -26861.49,E2 -26861.49} C_VEL
LIN {X 0,Y 117.419,Z 506.159,A -85,B 0,C 180,E1 -26865.911,E2 -26865.911} C_VEL
LIN {X 0,Y 117.774,Z 512.718,A -85,B 0,C 180,E1 -26870.875,E2 -26870.875} C_VEL
LIN {X 0,Y 117.655,Z 514.439,A -85,B 0,C 180,E1 -26872.155,E2 -26872.155} C_VEL
LIN {X 0,Y 112.111,Z 523.159,A -85,B 0,C 180,E1 -26876.735,E2 -26876.735} C_VEL
LIN {X 0,Y 107.286,Z 530.015,A -85,B 0,C 180,E1 -26881.646,E2 -26881.646} C_VEL
LIN {X 0,Y 102.629,Z 536.268,A -85,B 0,C 180,E1 -26887.875,E2 -26887.875} C_VEL
LIN {X 0,Y 99.41,Z 540.406,A -85,B 0,C 180,E1 -26893.574,E2 -26893.574} C_VEL
LIN {X 0,Y 97.565,Z 542.633,A -85,B 0,C 180,E1 -26897.521,E2 -26897.521} C_VEL
LIN {X 0,Y 96.3,Z 544.378,A -85,B 0,C 180,E1 -26901.608,E2 -26901.608} C_VEL
LIN {X 0,Y 95.373,Z 545.711,A -85,B 0,C 180,E1 -26905.775,E2 -26905.775} C_VEL
LIN {X 0,Y 95.138,Z 547.198,A -85,B 0,C 180,E1 -26914.237,E2 -26914.237} C_VEL
LIN {X 0,Y 95.471,Z 547.374,A -85,B 0,C 180,E1 -26918.467,E2 -26918.467} C_VEL
LIN {X 0,Y 96.167,Z 547.167,A -85,B 0,C 180,E1 -26922.666,E2 -26922.666} C_VEL
LIN {X 0,Y 99.563,Z 545.523,A -85,B 0,C 180,E1 -26930.668,E2 -26930.668} C_VEL
LIN {X 0,Y 101.83,Z 544.088,A -85,B 0,C 180,E1 -26934.464,E2 -26934.464} C_VEL
LIN {X 0,Y 105.864,Z 540.951,A -85,B 0,C 180,E1 -26940.34,E2 -26940.34} C_VEL
LIN {X 0,Y 111.72,Z 535.738,A -85,B 0,C 180,E1 -26946.701,E2 -26946.701} C_VEL
LIN {X 0,Y 117.053,Z 530.284,A -85,B 0,C 180,E1 -26951.335,E2 -26951.335} C_VEL
LIN {X 0,Y 121.974,Z 524.67,A -85,B 0,C 180,E1 -26954.878,E2 -26954.878} C_VEL
LIN {X 0,Y 122.791,Z 523.482,A -85,B 0,C 180,E1 -26955.64,E2 -26955.64} C_VEL
LIN {X 0,Y 123.412,Z 518.642,A -85,B 0,C 180,E1 -26960.193,E2 -26960.193} C_VEL
LIN {X 0,Y 123.474,Z 513.362,A -85,B 0,C 180,E1 -26965.306,E2 -26965.306} C_VEL
LIN {X 0,Y 123.188,Z 508.402,A -85,B 0,C 180,E1 -26970.418,E2 -26970.418} C_VEL
LIN {X 0,Y 122.903,Z 506.3,A -85,B 0,C 180,E1 -26972.775,E2 -26972.775} C_VEL
LIN {X 0,Y 122.445,Z 505.186,A -85,B 0,C 180,E1 -26974.501,E2 -26974.501} C_VEL
LIN {X 0,Y 120.37,Z 506.388,A -85,B 0,C 180,E1 -26975.876,E2 -26975.876} C_VEL
LIN {X 0,Y 113.439,Z 511.467,A -85,B 0,C 180,E1 -26980.077,E2 -26980.077} C_VEL
LIN {X 0,Y 110.005,Z 513.669,A -85,B 0,C 180,E1 -26983.404,E2 -26983.404} C_VEL
LIN {X 0,Y 106.443,Z 516.521,A -85,B 0,C 180,E1 -26986.638,E2 -26986.638} C_VEL
LIN {X 0,Y 104.972,Z 517.735,A -85,B 0,C 180,E1 -26988.412,E2 -26988.412} C_VEL
LIN {X 0,Y 102.891,Z 519.519,A -85,B 0,C 180,E1 -26992.148,E2 -26992.148} C_VEL
LIN {X 0,Y 100.524,Z 522.019,A -85,B 0,C 180,E1 -26995.99,E2 -26995.99} C_VEL
LIN {X 0,Y 98.644,Z 525.585,A -85,B 0,C 180,E1 -27004.085,E2 -27004.085} C_VEL
LIN {X 0,Y 98.038,Z 527.764,A -85,B 0,C 180,E1 -27008.242,E2 -27008.242} C_VEL
LIN {X 0,Y 98.657,Z 529.208,A -85,B 0,C 180,E1 -27012.339,E2 -27012.339} C_VEL
LIN {X 0,Y 99.239,Z 531.169,A -85,B 0,C 180,E1 -27016.455,E2 -27016.455} C_VEL
LIN {X 0,Y 100.683,Z 532.775,A -85,B 0,C 180,E1 -27020.427,E2 -27020.427} C_VEL
LIN {X 0,Y 102.732,Z 533.325,A -85,B 0,C 180,E1 -27023.163,E2 -27023.163} C_VEL
LIN {X 0,Y 110.207,Z 542.359,A -85,B 0,C 180,E1 -27030.674,E2 -27030.674} C_VEL
LIN {X 0,Y 118.395,Z 548.97,A -85,B 0,C 180,E1 -27036.413,E2 -27036.413} C_VEL
LIN {X 0,Y 124.67,Z 552.724,A -85,B 0,C 180,E1 -27039.777,E2 -27039.777} C_VEL
LIN {X 0,Y 125.084,Z 553.342,A -85,B 0,C 180,E1 -27040.79,E2 -27040.79} C_VEL
LIN {X 0,Y 114.35,Z 552.508,A -85,B 0,C 180,E1 -27047.716,E2 -27047.716} C_VEL
LIN {X 0,Y 107.927,Z 558.547,A -85,B 0,C 180,E1 -27051.783,E2 -27051.783} C_VEL
LIN {X 0,Y 102.237,Z 563.604,A -85,B 0,C 180,E1 -27056.636,E2 -27056.636} C_VEL
LIN {X 0,Y 97.905,Z 567.622,A -85,B 0,C 180,E1 -27062.186,E2 -27062.186} C_VEL
LIN {X 0,Y 94.843,Z 570.667,A -85,B 0,C 180,E1 -27068.252,E2 -27068.252} C_VEL
LIN {X 0,Y 92.82,Z 573.297,A -85,B 0,C 180,E1 -27076.87,E2 -27076.87} C_VEL
LIN {X 0,Y 92.723,Z 574.049,A -85,B 0,C 180,E1 -27081.28,E2 -27081.28} C_VEL
LIN {X 0,Y 93.176,Z 574.376,A -85,B 0,C 180,E1 -27085.673,E2 -27085.673} C_VEL
LIN {X 0,Y 93.852,Z 574.265,A -85,B 0,C 180,E1 -27089.999,E2 -27089.999} C_VEL
LIN {X 0,Y 93.08,Z 573.484,A -85,B 0,C 180,E1 -27094.329,E2 -27094.329} C_VEL
LIN {X 0,Y 92.662,Z 571.984,A -85,B 0,C 180,E1 -27099.602,E2 -27099.602} C_VEL
LIN {X 0,Y 93.326,Z 568.534,A -85,B 0,C 180,E1 -27107.53,E2 -27107.53} C_VEL
LIN {X 0,Y 95.262,Z 564.554,A -85,B 0,C 180,E1 -27113.938,E2 -27113.938} C_VEL
LIN {X 0,Y 98.541,Z 559.485,A -85,B 0,C 180,E1 -27119.949,E2 -27119.949} C_VEL
LIN {X 0,Y 101.792,Z 554.247,A -85,B 0,C 180,E1 -27124.722,E2 -27124.722} C_VEL
LIN {X 0,Y 105.723,Z 546.407,A -85,B 0,C 180,E1 -27130.4,E2 -27130.4} C_VEL
LIN {X 0,Y 109.511,Z 538.153,A -85,B 0,C 180,E1 -27135.095,E2 -27135.095} C_VEL
LIN {X 0,Y 113.16,Z 528.646,A -85,B 0,C 180,E1 -27139.535,E2 -27139.535} C_VEL
LIN {X 0,Y 116.334,Z 518.132,A -85,B 0,C 180,E1 -27143.669,E2 -27143.669} C_VEL
LIN {X 0,Y 117.841,Z 511.517,A -85,B 0,C 180,E1 -27146.022,E2 -27146.022} C_VEL
LIN {X 0,Y 116.648,Z 503.412,A -85,B 0,C 180,E1 -27150.485,E2 -27150.485} C_VEL
LIN {X 0,Y 115.228,Z 496.488,A -85,B 0,C 180,E1 -27154.727,E2 -27154.727} C_VEL
LIN {X 0,Y 113.888,Z 491.488,A -85,B 0,C 180,E1 -27158.269,E2 -27158.269} C_VEL
LIN {X 0,Y 111.953,Z 485.345,A -85,B 0,C 180,E1 -27163.591,E2 -27163.591} C_VEL
LIN {X 0,Y 110.763,Z 482.29,A -85,B 0,C 180,E1 -27167.169,E2 -27167.169} C_VEL
LIN {X 0,Y 109.461,Z 478.323,A -85,B 0,C 180,E1 -27172.623,E2 -27172.623} C_VEL
LIN {X 0,Y 108.644,Z 477.169,A -85,B 0,C 180,E1 -27176.292,E2 -27176.292} C_VEL
LIN {X 0,Y 108.093,Z 476.566,A -85,B 0,C 180,E1 -27180.001,E2 -27180.001} C_VEL
LIN {X 0,Y 107.841,Z 476.863,A -85,B 0,C 180,E1 -27187.49,E2 -27187.49} C_VEL
LIN {X 0,Y 108.217,Z 477.369,A -85,B 0,C 180,E1 -27191.235,E2 -27191.235} C_VEL
LIN {X 0,Y 110.426,Z 482.712,A -85,B 0,C 180,E1 -27202.45,E2 -27202.45} C_VEL
LIN {X 0,Y 112.507,Z 487.542,A -85,B 0,C 180,E1 -27209.011,E2 -27209.011} C_VEL
LIN {X 0,Y 114.115,Z 491.818,A -85,B 0,C 180,E1 -27213.662,E2 -27213.662} C_VEL
LIN {X 0,Y 115.615,Z 497,A -85,B 0,C 180,E1 -27218.43,E2 -27218.43} C_VEL
LIN {X 0,Y 116.515,Z 500.558,A -85,B 0,C 180,E1 -27221.49,E2 -27221.49} C_VEL
LIN {X 0,Y 116.423,Z 502.954,A -85,B 0,C 180,E1 -27223.032,E2 -27223.032} C_VEL
LIN {X 0,Y 115.123,Z 506.707,A -85,B 0,C 180,E1 -27224.783,E2 -27224.783} C_VEL
LIN {X 0,Y 112.472,Z 512.427,A -85,B 0,C 180,E1 -27227.43,E2 -27227.43} C_VEL
LIN {X 0,Y 111.799,Z 514.871,A -85,B 0,C 180,E1 -27229.052,E2 -27229.052} C_VEL
LIN {X 0,Y 111.676,Z 516.446,A -85,B 0,C 180,E1 -27230.337,E2 -27230.337} C_VEL
LIN {X 0,Y 106.32,Z 524.313,A -85,B 0,C 180,E1 -27234.663,E2 -27234.663} C_VEL
LIN {X 0,Y 101.171,Z 531.134,A -85,B 0,C 180,E1 -27239.76,E2 -27239.76} C_VEL
LIN {X 0,Y 96.172,Z 537.365,A -85,B 0,C 180,E1 -27246.302,E2 -27246.302} C_VEL
LIN {X 0,Y 92.712,Z 541.482,A -85,B 0,C 180,E1 -27252.35,E2 -27252.35} C_VEL
LIN {X 0,Y 90.728,Z 543.701,A -85,B 0,C 180,E1 -27256.563,E2 -27256.563} C_VEL
LIN {X 0,Y 89.363,Z 545.428,A -85,B 0,C 180,E1 -27260.951,E2 -27260.951} C_VEL
LIN {X 0,Y 88.368,Z 546.754,A -85,B 0,C 180,E1 -27265.439,E2 -27265.439} C_VEL
LIN {X 0,Y 88.129,Z 548.222,A -85,B 0,C 180,E1 -27274.575,E2 -27274.575} C_VEL
LIN {X 0,Y 88.522,Z 548.382,A -85,B 0,C 180,E1 -27279.137,E2 -27279.137} C_VEL
LIN {X 0,Y 89.318,Z 548.167,A -85,B 0,C 180,E1 -27283.655,E2 -27283.655} C_VEL
LIN {X 0,Y 93.019,Z 546.504,A -85,B 0,C 180,E1 -27292.197,E2 -27292.197} C_VEL
LIN {X 0,Y 95.473,Z 545.052,A -85,B 0,C 180,E1 -27296.212,E2 -27296.212} C_VEL
LIN {X 0,Y 99.807,Z 541.933,A -85,B 0,C 180,E1 -27302.327,E2 -27302.327} C_VEL
LIN {X 0,Y 104.394,Z 538.224,A -85,B 0,C 180,E1 -27307.295,E2 -27307.295} C_VEL
LIN {X 0,Y 109.864,Z 533.149,A -85,B 0,C 180,E1 -27312.199,E2 -27312.199} C_VEL
LIN {X 0,Y 116.057,Z 526.725,A -85,B 0,C 180,E1 -27316.61,E2 -27316.61} C_VEL
LIN {X 0,Y 116.877,Z 525.457,A -85,B 0,C 180,E1 -27317.592,E2 -27317.592} C_VEL
LIN {X 0,Y 117.651,Z 520.834,A -85,B 0,C 180,E1 -27322.442,E2 -27322.442} C_VEL
LIN {X 0,Y 117.929,Z 517.052,A -85,B 0,C 180,E1 -27326.548,E2 -27326.548} C_VEL
LIN {X 0,Y 118.023,Z 512.673,A -85,B 0,C 180,E1 -27331.55,E2 -27331.55} C_VEL
LIN {X 0,Y 117.937,Z 511.216,A -85,B 0,C 180,E1 -27333.366,E2 -27333.366} C_VEL
LIN {X 0,Y 117.46,Z 511.339,A -85,B 0,C 180,E1 -27333.833,E2 -27333.833} C_VEL
LIN {X 0,Y 110.655,Z 515.847,A -85,B 0,C 180,E1 -27337.599,E2 -27337.599} C_VEL
LIN {X 0,Y 104.911,Z 519.352,A -85,B 0,C 180,E1 -27342.573,E2 -27342.573} C_VEL
LIN {X 0,Y 101.573,Z 521.793,A -85,B 0,C 180,E1 -27345.627,E2 -27345.627} C_VEL
LIN {X 0,Y 97.547,Z 524.862,A -85,B 0,C 180,E1 -27351.714,E2 -27351.714} C_VEL
LIN {X 0,Y 95.247,Z 527.134,A -85,B 0,C 180,E1 -27355.768,E2 -27355.768} C_VEL
LIN {X 0,Y 92.723,Z 532.627,A -85,B 0,C 180,E1 -27368.718,E2 -27368.718} C_VEL
LIN {X 0,Y 93.265,Z 534.163,A -85,B 0,C 180,E1 -27373.065,E2 -27373.065} C_VEL
LIN {X 0,Y 94.008,Z 535.991,A -85,B 0,C 180,E1 -27377.399,E2 -27377.399} C_VEL
LIN {X 0,Y 100.548,Z 540.248,A -85,B 0,C 180,E1 -27389.293,E2 -27389.293} C_VEL
LIN {X 0,Y 104.515,Z 541.142,A -85,B 0,C 180,E1 -27392.83,E2 -27392.83} C_VEL
LIN {X 0,Y 112.794,Z 547.98,A -85,B 0,C 180,E1 -27398.541,E2 -27398.541} C_VEL
LIN {X 0,Y 116.389,Z 550.323,A -85,B 0,C 180,E1 -27400.52,E2 -27400.52} C_VEL
LIN {X 0,Y 115.305,Z 550.354,A -85,B 0,C 180,E1 -27401.501,E2 -27401.501} C_VEL
LIN {X 0,Y 111.091,Z 549.882,A -85,B 0,C 180,E1 -27404.302,E2 -27404.302} C_VEL
LIN {X 0,Y 104.705,Z 555.675,A -85,B 0,C 180,E1 -27407.837,E2 -27407.837} C_VEL
LIN {X 0,Y 98.304,Z 561.106,A -85,B 0,C 180,E1 -27412.576,E2 -27412.576} C_VEL
LIN {X 0,Y 93.122,Z 565.437,A -85,B 0,C 180,E1 -27418.108,E2 -27418.108} C_VEL
LIN {X 0,Y 90.349,Z 567.781,A -85,B 0,C 180,E1 -27422.177,E2 -27422.177} C_VEL
LIN {X 0,Y 86.753,Z 571.172,A -85,B 0,C 180,E1 -27431.091,E2 -27431.091} C_VEL
LIN {X 0,Y 85.676,Z 573.031,A -85,B 0,C 180,E1 -27440.556,E2 -27440.556} C_VEL
LIN {X 0,Y 86.066,Z 573.345,A -85,B 0,C 180,E1 -27445.315,E2 -27445.315} C_VEL
LIN {X 0,Y 86.736,Z 573.228,A -85,B 0,C 180,E1 -27449.999,E2 -27449.999} C_VEL
LIN {X 0,Y 85.97,Z 572.436,A -85,B 0,C 180,E1 -27454.688,E2 -27454.688} C_VEL
LIN {X 0,Y 85.618,Z 571.075,A -85,B 0,C 180,E1 -27459.931,E2 -27459.931} C_VEL
LIN {X 0,Y 86.505,Z 567.444,A -85,B 0,C 180,E1 -27468.963,E2 -27468.963} C_VEL
LIN {X 0,Y 88.753,Z 563.446,A -85,B 0,C 180,E1 -27475.817,E2 -27475.817} C_VEL
LIN {X 0,Y 92.416,Z 558.362,A -85,B 0,C 180,E1 -27482.162,E2 -27482.162} C_VEL
LIN {X 0,Y 95.809,Z 553.063,A -85,B 0,C 180,E1 -27487.24,E2 -27487.24} C_VEL
LIN {X 0,Y 100.196,Z 545.195,A -85,B 0,C 180,E1 -27493.147,E2 -27493.147} C_VEL
LIN {X 0,Y 104.153,Z 537.132,A -85,B 0,C 180,E1 -27497.922,E2 -27497.922} C_VEL
LIN {X 0,Y 108.154,Z 527.608,A -85,B 0,C 180,E1 -27502.53,E2 -27502.53} C_VEL
LIN {X 0,Y 111.785,Z 516.681,A -85,B 0,C 180,E1 -27506.968,E2 -27506.968} C_VEL
LIN {X 0,Y 112.36,Z 513.941,A -85,B 0,C 180,E1 -27508.102,E2 -27508.102} C_VEL
LIN {X 0,Y 111.571,Z 506.406,A -85,B 0,C 180,E1 -27512.727,E2 -27512.727} C_VEL
LIN {X 0,Y 110.642,Z 500.492,A -85,B 0,C 180,E1 -27516.755,E2 -27516.755} C_VEL
LIN {X 0,Y 109.363,Z 495.001,A -85,B 0,C 180,E1 -27521.258,E2 -27521.258} C_VEL
LIN {X 0,Y 108.485,Z 490.919,A -85,B 0,C 180,E1 -27524.982,E2 -27524.982} C_VEL
LIN {X 0,Y 107.155,Z 486.672,A -85,B 0,C 180,E1 -27530.563,E2 -27530.563} C_VEL
LIN {X 0,Y 106.862,Z 485.369,A -85,B 0,C 180,E1 -27532.442,E2 -27532.442} C_VEL
LIN {X 0,Y 106.169,Z 483.873,A -85,B 0,C 180,E1 -27536.205,E2 -27536.205} C_VEL
LIN {X 0,Y 105.442,Z 483.242,A -85,B 0,C 180,E1 -27541.204,E2 -27541.204} C_VEL
LIN {X 0,Y 105.206,Z 483.49,A -85,B 0,C 180,E1 -27547.679,E2 -27547.679} C_VEL
LIN {X 0,Y 105.459,Z 484.158,A -85,B 0,C 180,E1 -27551.533,E2 -27551.533} C_VEL
LIN {X 0,Y 106.795,Z 488.481,A -85,B 0,C 180,E1 -27561.221,E2 -27561.221} C_VEL
LIN {X 0,Y 108.182,Z 492.228,A -85,B 0,C 180,E1 -27567.05,E2 -27567.05} C_VEL
LIN {X 0,Y 109.179,Z 495.387,A -85,B 0,C 180,E1 -27570.996,E2 -27570.996} C_VEL
LIN {X 0,Y 110.413,Z 500.625,A -85,B 0,C 180,E1 -27576.468,E2 -27576.468} C_VEL
LIN {X 0,Y 111.381,Z 505.977,A -85,B 0,C 180,E1 -27581.492,E2 -27581.492} C_VEL
LIN {X 0,Y 111.768,Z 511.532,A -85,B 0,C 180,E1 -27586.237,E2 -27586.237} C_VEL
LIN {X 0,Y 111.799,Z 514.871,A -85,B 0,C 180,E1 -27589.052,E2 -27589.052} C_VEL
LIN {X 0,Y 111.005,Z 517.205,A -85,B 0,C 180,E1 -27590.574,E2 -27590.574} C_VEL
LIN {X 0,Y 109.324,Z 519.669,A -85,B 0,C 180,E1 -27591.834,E2 -27591.834} C_VEL
LIN {X 0,Y 107.043,Z 522.206,A -85,B 0,C 180,E1 -27592.914,E2 -27592.914} C_VEL
LIN {X 0,Y 97.263,Z 530.591,A -85,B 0,C 180,E1 -27596.613,E2 -27596.613} C_VEL
LIN {X 0,Y 94.356,Z 533.257,A -85,B 0,C 180,E1 -27598.614,E2 -27598.614} C_VEL
LIN {X 0,Y 93.903,Z 533.747,A -85,B 0,C 180,E1 -27599.093,E2 -27599.093} C_VEL
LIN {X 0,Y 89.796,Z 538.461,A -85,B 0,C 180,E1 -27604.504,E2 -27604.504} C_VEL
LIN {X 0,Y 86.06,Z 542.558,A -85,B 0,C 180,E1 -27610.935,E2 -27610.935} C_VEL
LIN {X 0,Y 83.94,Z 544.764,A -85,B 0,C 180,E1 -27615.454,E2 -27615.454} C_VEL
LIN {X 0,Y 82.439,Z 546.477,A -85,B 0,C 180,E1 -27620.184,E2 -27620.184} C_VEL
LIN {X 0,Y 81.367,Z 547.796,A -85,B 0,C 180,E1 -27625.046,E2 -27625.046} C_VEL
LIN {X 0,Y 81.124,Z 549.245,A -85,B 0,C 180,E1 -27634.971,E2 -27634.971} C_VEL
LIN {X 0,Y 81.588,Z 549.391,A -85,B 0,C 180,E1 -27639.922,E2 -27639.922} C_VEL
LIN {X 0,Y 82.501,Z 549.167,A -85,B 0,C 180,E1 -27644.808,E2 -27644.808} C_VEL
LIN {X 0,Y 86.55,Z 547.484,A -85,B 0,C 180,E1 -27653.955,E2 -27653.955} C_VEL
LIN {X 0,Y 89.217,Z 546.016,A -85,B 0,C 180,E1 -27658.207,E2 -27658.207} C_VEL
LIN {X 0,Y 93.889,Z 542.912,A -85,B 0,C 180,E1 -27664.572,E2 -27664.572} C_VEL
LIN {X 0,Y 98.89,Z 539.149,A -85,B 0,C 180,E1 -27669.765,E2 -27669.765} C_VEL
LIN {X 0,Y 104.753,Z 534.054,A -85,B 0,C 180,E1 -27674.787,E2 -27674.787} C_VEL
LIN {X 0,Y 110.201,Z 528.808,A -85,B 0,C 180,E1 -27678.536,E2 -27678.536} C_VEL
LIN {X 0,Y 110.983,Z 527.674,A -85,B 0,C 180,E1 -27679.457,E2 -27679.457} C_VEL
LIN {X 0,Y 112.007,Z 523.285,A -85,B 0,C 180,E1 -27684.658,E2 -27684.658} C_VEL
LIN {X 0,Y 112.542,Z 518.938,A -85,B 0,C 180,E1 -27690.027,E2 -27690.027} C_VEL
LIN {X 0,Y 112.449,Z 517.261,A -85,B 0,C 180,E1 -27692.572,E2 -27692.572} C_VEL
LIN {X 0,Y 107.873,Z 519.981,A -85,B 0,C 180,E1 -27694.943,E2 -27694.943} C_VEL
LIN {X 0,Y 101.701,Z 523.362,A -85,B 0,C 180,E1 -27699.786,E2 -27699.786} C_VEL
LIN {X 0,Y 97.586,Z 525.97,A -85,B 0,C 180,E1 -27703.257,E2 -27703.257} C_VEL
LIN {X 0,Y 89.693,Z 531.942,A -85,B 0,C 180,E1 -27715.505,E2 -27715.505} C_VEL
LIN {X 0,Y 87.182,Z 537.171,A -85,B 0,C 180,E1 -27729.277,E2 -27729.277} C_VEL
LIN {X 0,Y 88.598,Z 540.467,A -85,B 0,C 180,E1 -27738.499,E2 -27738.499} C_VEL
LIN {X 0,Y 95.64,Z 544.535,A -85,B 0,C 180,E1 -27750.956,E2 -27750.956} C_VEL
LIN {X 0,Y 99.391,Z 545.46,A -85,B 0,C 180,E1 -27754.449,E2 -27754.449} C_VEL
LIN {X 0,Y 102.907,Z 546.9,A -85,B 0,C 180,E1 -27757.926,E2 -27757.926} C_VEL
LIN {X 0,Y 107.342,Z 547.811,A -85,B 0,C 180,E1 -27760.899,E2 -27760.899} C_VEL
LIN {X 0,Y 99.578,Z 554.76,A -85,B 0,C 180,E1 -27765.106,E2 -27765.106} C_VEL
LIN {X 0,Y 92.791,Z 560.171,A -85,B 0,C 180,E1 -27769.923,E2 -27769.923} C_VEL
LIN {X 0,Y 87.179,Z 564.479,A -85,B 0,C 180,E1 -27775.644,E2 -27775.644} C_VEL
LIN {X 0,Y 84.129,Z 566.808,A -85,B 0,C 180,E1 -27779.917,E2 -27779.917} C_VEL
LIN {X 0,Y 80.044,Z 570.175,A -85,B 0,C 180,E1 -27789.438,E2 -27789.438} C_VEL
LIN {X 0,Y 78.643,Z 572.01,A -85,B 0,C 180,E1 -27799.703,E2 -27799.703} C_VEL
LIN {X 0,Y 78.948,Z 572.312,A -85,B 0,C 180,E1 -27804.892,E2 -27804.892} C_VEL
LIN {X 0,Y 79.617,Z 572.19,A -85,B 0,C 180,E1 -27809.999,E2 -27809.999} C_VEL
LIN {X 0,Y 78.864,Z 571.388,A -85,B 0,C 180,E1 -27815.112,E2 -27815.112} C_VEL
LIN {X 0,Y 78.574,Z 570.164,A -85,B 0,C 180,E1 -27820.304,E2 -27820.304} C_VEL
LIN {X 0,Y 79.218,Z 567.488,A -85,B 0,C 180,E1 -27828.089,E2 -27828.089} C_VEL
LIN {X 0,Y 81.303,Z 563.811,A -85,B 0,C 180,E1 -27835.607,E2 -27835.607} C_VEL
LIN {X 0,Y 84.936,Z 559.091,A -85,B 0,C 180,E1 -27842.536,E2 -27842.536} C_VEL
LIN {X 0,Y 88.475,Z 554.403,A -85,B 0,C 180,E1 -27847.679,E2 -27847.679} C_VEL
LIN {X 0,Y 93.2,Z 546.826,A -85,B 0,C 180,E1 -27854.227,E2 -27854.227} C_VEL
LIN {X 0,Y 96.975,Z 540.202,A -85,B 0,C 180,E1 -27858.662,E2 -27858.662} C_VEL
LIN {X 0,Y 101.929,Z 530.174,A -85,B 0,C 180,E1 -27864.11,E2 -27864.11} C_VEL
LIN {X 0,Y 105.927,Z 520.121,A -85,B 0,C 180,E1 -27868.609,E2 -27868.609} C_VEL
LIN {X 0,Y 106.934,Z 516.988,A -85,B 0,C 180,E1 -27869.946,E2 -27869.946} C_VEL
LIN {X 0,Y 106.597,Z 510.04,A -85,B 0,C 180,E1 -27874.625,E2 -27874.625} C_VEL
LIN {X 0,Y 106.049,Z 504.766,A -85,B 0,C 180,E1 -27878.622,E2 -27878.622} C_VEL
LIN {X 0,Y 105.346,Z 500.314,A -85,B 0,C 180,E1 -27882.53,E2 -27882.53} C_VEL
LIN {X 0,Y 104.775,Z 496.371,A -85,B 0,C 180,E1 -27886.423,E2 -27886.423} C_VEL
LIN {X 0,Y 103.814,Z 492.265,A -85,B 0,C 180,E1 -27892.219,E2 -27892.219} C_VEL
LIN {X 0,Y 103.293,Z 490.484,A -85,B 0,C 180,E1 -27896.099,E2 -27896.099} C_VEL
LIN {X 0,Y 102.746,Z 489.722,A -85,B 0,C 180,E1 -27900.001,E2 -27900.001} C_VEL
LIN {X 0,Y 102.212,Z 489.97,A -85,B 0,C 180,E1 -27907.905,E2 -27907.905} C_VEL
LIN {X 0,Y 102.31,Z 490.839,A -85,B 0,C 180,E1 -27911.893,E2 -27911.893} C_VEL
LIN {X 0,Y 102.964,Z 494.157,A -85,B 0,C 180,E1 -27919.956,E2 -27919.956} C_VEL
LIN {X 0,Y 103.978,Z 497.644,A -85,B 0,C 180,E1 -27926.063,E2 -27926.063} C_VEL
LIN {X 0,Y 104.671,Z 500.718,A -85,B 0,C 180,E1 -27930.236,E2 -27930.236} C_VEL
LIN {X 0,Y 105.39,Z 505.149,A -85,B 0,C 180,E1 -27935.321,E2 -27935.321} C_VEL
LIN {X 0,Y 105.932,Z 509.922,A -85,B 0,C 180,E1 -27940.305,E2 -27940.305} C_VEL
LIN {X 0,Y 106.022,Z 514.387,A -85,B 0,C 180,E1 -27944.551,E2 -27944.551} C_VEL
LIN {X 0,Y 105.763,Z 518.529,A -85,B 0,C 180,E1 -27948.357,E2 -27948.357} C_VEL
LIN {X 0,Y 99.717,Z 526.675,A -85,B 0,C 180,E1 -27953.197,E2 -27953.197} C_VEL
LIN {X 0,Y 94.355,Z 533.232,A -85,B 0,C 180,E1 -27958.575,E2 -27958.575} C_VEL
LIN {X 0,Y 93.903,Z 533.747,A -85,B 0,C 180,E1 -27959.093,E2 -27959.093} C_VEL
LIN {X 0,Y 90.986,Z 536.557,A -85,B 0,C 180,E1 -27961.778,E2 -27961.778} C_VEL
LIN {X 0,Y 84.92,Z 540.86,A -85,B 0,C 180,E1 -27966.069,E2 -27966.069} C_VEL
LIN {X 0,Y 79.153,Z 544.455,A -85,B 0,C 180,E1 -27971.142,E2 -27971.142} C_VEL
LIN {X 0,Y 76.875,Z 546.104,A -85,B 0,C 180,E1 -27974.97,E2 -27974.97} C_VEL
LIN {X 0,Y 74.37,Z 548.838,A -85,B 0,C 180,E1 -27984.579,E2 -27984.579} C_VEL
LIN {X 0,Y 74.124,Z 550.265,A -85,B 0,C 180,E1 -27995.442,E2 -27995.442} C_VEL
LIN {X 0,Y 75.722,Z 550.167,A -85,B 0,C 180,E1 -28006.168,E2 -28006.168} C_VEL
LIN {X 0,Y 80.177,Z 548.462,A -85,B 0,C 180,E1 -28015.996,E2 -28015.996} C_VEL
LIN {X 0,Y 83.085,Z 546.981,A -85,B 0,C 180,E1 -28020.501,E2 -28020.501} C_VEL
LIN {X 0,Y 88.143,Z 543.886,A -85,B 0,C 180,E1 -28027.121,E2 -28027.121} C_VEL
LIN {X 0,Y 93.591,Z 540.075,A -85,B 0,C 180,E1 -28032.521,E2 -28032.521} C_VEL
LIN {X 0,Y 99.878,Z 534.959,A -85,B 0,C 180,E1 -28037.634,E2 -28037.634} C_VEL
LIN {X 0,Y 104.484,Z 530.816,A -85,B 0,C 180,E1 -28040.674,E2 -28040.674} C_VEL
LIN {X 0,Y 105.289,Z 529.57,A -85,B 0,C 180,E1 -28041.974,E2 -28041.974} C_VEL
LIN {X 0,Y 106.169,Z 526.716,A -85,B 0,C 180,E1 -28045.759,E2 -28045.759} C_VEL
LIN {X 0,Y 106.962,Z 523.122,A -85,B 0,C 180,E1 -28050.786,E2 -28050.786} C_VEL
LIN {X 0,Y 105.144,Z 523.855,A -85,B 0,C 180,E1 -28052.102,E2 -28052.102} C_VEL
LIN {X 0,Y 96.108,Z 528.448,A -85,B 0,C 180,E1 -28058.553,E2 -28058.553} C_VEL
LIN {X 0,Y 92.088,Z 530.679,A -85,B 0,C 180,E1 -28062.225,E2 -28062.225} C_VEL
LIN {X 0,Y 83.854,Z 536.381,A -85,B 0,C 180,E1 -28075.191,E2 -28075.191} C_VEL
LIN {X 0,Y 81.845,Z 543.031,A -85,B 0,C 180,E1 -28094.927,E2 -28094.927} C_VEL
LIN {X 0,Y 85.101,Z 546.01,A -85,B 0,C 180,E1 -28104.709,E2 -28104.709} C_VEL
LIN {X 0,Y 90.625,Z 548.513,A -85,B 0,C 180,E1 -28112.877,E2 -28112.877} C_VEL
LIN {X 0,Y 94.496,Z 549.512,A -85,B 0,C 180,E1 -28116.511,E2 -28116.511} C_VEL
LIN {X 0,Y 98.315,Z 550.845,A -85,B 0,C 180,E1 -28120.042,E2 -28120.042} C_VEL
LIN {X 0,Y 89.828,Z 557.592,A -85,B 0,C 180,E1 -28125.238,E2 -28125.238} C_VEL
LIN {X 0,Y 83.269,Z 562.213,A -85,B 0,C 180,E1 -28130.726,E2 -28130.726} C_VEL
LIN {X 0,Y 78.067,Z 565.834,A -85,B 0,C 180,E1 -28137.304,E2 -28137.304} C_VEL
LIN {X 0,Y 73.408,Z 569.177,A -85,B 0,C 180,E1 -28147.482,E2 -28147.482} C_VEL
LIN {X 0,Y 71.624,Z 570.988,A -85,B 0,C 180,E1 -28158.681,E2 -28158.681} C_VEL
LIN {X 0,Y 71.842,Z 571.28,A -85,B 0,C 180,E1 -28164.385,E2 -28164.385} C_VEL
LIN {X 0,Y 72.496,Z 571.153,A -85,B 0,C 180,E1 -28169.999,E2 -28169.999} C_VEL
LIN {X 0,Y 71.744,Z 570.337,A -85,B 0,C 180,E1 -28175.62,E2 -28175.62} C_VEL
LIN {X 0,Y 71.512,Z 569.094,A -85,B 0,C 180,E1 -28181.334,E2 -28181.334} C_VEL
LIN {X 0,Y 72.423,Z 566.405,A -85,B 0,C 180,E1 -28189.854,E2 -28189.854} C_VEL
LIN {X 0,Y 74.899,Z 562.713,A -85,B 0,C 180,E1 -28197.979,E2 -28197.979} C_VEL
LIN {X 0,Y 78.992,Z 557.974,A -85,B 0,C 180,E1 -28205.331,E2 -28205.331} C_VEL
LIN {X 0,Y 82.532,Z 553.574,A -85,B 0,C 180,E1 -28210.432,E2 -28210.432} C_VEL
LIN {X 0,Y 88.028,Z 545.62,A -85,B 0,C 180,E1 -28217.603,E2 -28217.603} C_VEL
LIN {X 0,Y 93.314,Z 536.902,A -85,B 0,C 180,E1 -28223.453,E2 -28223.453} C_VEL
LIN {X 0,Y 98.057,Z 527.772,A -85,B 0,C 180,E1 -28228.332,E2 -28228.332} C_VEL
LIN {X 0,Y 101.518,Z 519.63,A -85,B 0,C 180,E1 -28232.143,E2 -28232.143} C_VEL
LIN {X 0,Y 101.574,Z 513.352,A -85,B 0,C 180,E1 -28236.833,E2 -28236.833} C_VEL
LIN {X 0,Y 101.377,Z 508.697,A -85,B 0,C 180,E1 -28240.774,E2 -28240.774} C_VEL
LIN {X 0,Y 101.097,Z 505.471,A -85,B 0,C 180,E1 -28243.856,E2 -28243.856} C_VEL
LIN {X 0,Y 100.849,Z 501.649,A -85,B 0,C 180,E1 -28247.933,E2 -28247.933} C_VEL
LIN {X 0,Y 100.366,Z 498.945,A -85,B 0,C 180,E1 -28251.95,E2 -28251.95} C_VEL
LIN {X 0,Y 99.981,Z 496.959,A -85,B 0,C 180,E1 -28255.97,E2 -28255.97} C_VEL
LIN {X 0,Y 99.494,Z 496.044,A -85,B 0,C 180,E1 -28260.001,E2 -28260.001} C_VEL
LIN {X 0,Y 98.847,Z 496.317,A -85,B 0,C 180,E1 -28268.176,E2 -28268.176} C_VEL
LIN {X 0,Y 98.759,Z 497.295,A -85,B 0,C 180,E1 -28272.328,E2 -28272.328} C_VEL
LIN {X 0,Y 99.105,Z 500.668,A -85,B 0,C 180,E1 -28280.768,E2 -28280.768} C_VEL
LIN {X 0,Y 99.592,Z 502.934,A -85,B 0,C 180,E1 -28285.051,E2 -28285.051} C_VEL
LIN {X 0,Y 100.152,Z 507.609,A -85,B 0,C 180,E1 -28291.759,E2 -28291.759} C_VEL
LIN {X 0,Y 100.413,Z 512.292,A -85,B 0,C 180,E1 -28297.333,E2 -28297.333} C_VEL
LIN {X 0,Y 100.387,Z 516.281,A -85,B 0,C 180,E1 -28301.687,E2 -28301.687} C_VEL
LIN {X 0,Y 99.896,Z 520.6,A -85,B 0,C 180,E1 -28306.145,E2 -28306.145} C_VEL
LIN {X 0,Y 94.196,Z 527.818,A -85,B 0,C 180,E1 -28310.641,E2 -28310.641} C_VEL
LIN {X 0,Y 88.048,Z 534.773,A -85,B 0,C 180,E1 -28316.653,E2 -28316.653} C_VEL
LIN {X 0,Y 83.521,Z 539.558,A -85,B 0,C 180,E1 -28322.433,E2 -28322.433} C_VEL
LIN {X 0,Y 79.467,Z 543.635,A -85,B 0,C 180,E1 -28329.284,E2 -28329.284} C_VEL
LIN {X 0,Y 76.875,Z 546.104,A -85,B 0,C 180,E1 -28334.97,E2 -28334.97} C_VEL
LIN {X 0,Y 74.927,Z 547.588,A -85,B 0,C 180,E1 -28339.047,E2 -28339.047} C_VEL
LIN {X 0,Y 70.812,Z 549.657,A -85,B 0,C 180,E1 -28345.949,E2 -28345.949} C_VEL
LIN {X 0,Y 68.094,Z 550.824,A -85,B 0,C 180,E1 -28352.034,E2 -28352.034} C_VEL
LIN {X 0,Y 67.258,Z 551.307,A -85,B 0,C 180,E1 -28356.98,E2 -28356.98} C_VEL
LIN {X 0,Y 67.327,Z 551.339,A -85,B 0,C 180,E1 -28358.658,E2 -28358.658} C_VEL
LIN {X 0,Y 68.995,Z 551.167,A -85,B 0,C 180,E1 -28367.795,E2 -28367.795} C_VEL
LIN {X 0,Y 71.136,Z 550.505,A -85,B 0,C 180,E1 -28373.279,E2 -28373.279} C_VEL
LIN {X 0,Y 73.922,Z 549.439,A -85,B 0,C 180,E1 -28378.385,E2 -28378.385} C_VEL
LIN {X 0,Y 77.107,Z 547.946,A -85,B 0,C 180,E1 -28383.154,E2 -28383.154} C_VEL
LIN {X 0,Y 82.619,Z 544.847,A -85,B 0,C 180,E1 -28390.039,E2 -28390.039} C_VEL
LIN {X 0,Y 88.534,Z 541.001,A -85,B 0,C 180,E1 -28395.599,E2 -28395.599} C_VEL
LIN {X 0,Y 95.277,Z 535.863,A -85,B 0,C 180,E1 -28400.763,E2 -28400.763} C_VEL
LIN {X 0,Y 99.006,Z 532.723,A -85,B 0,C 180,E1 -28403.111,E2 -28403.111} C_VEL
LIN {X 0,Y 99.967,Z 530.849,A -85,B 0,C 180,E1 -28405.775,E2 -28405.775} C_VEL
LIN {X 0,Y 100.33,Z 529.901,A -85,B 0,C 180,E1 -28407.204,E2 -28407.204} C_VEL
LIN {X 0,Y 99.897,Z 528.656,A -85,B 0,C 180,E1 -28410.496,E2 -28410.496} C_VEL
LIN {X 0,Y 92.817,Z 531.854,A -85,B 0,C 180,E1 -28415.319,E2 -28415.319} C_VEL
LIN {X 0,Y 90.365,Z 533.073,A -85,B 0,C 180,E1 -28417.115,E2 -28417.115} C_VEL
LIN {X 0,Y 77.781,Z 540.483,A -85,B 0,C 180,E1 -28434.815,E2 -28434.815} C_VEL
LIN {X 0,Y 75.882,Z 546.865,A -85,B 0,C 180,E1 -28456.131,E2 -28456.131} C_VEL
LIN {X 0,Y 79.391,Z 549.661,A -85,B 0,C 180,E1 -28466.271,E2 -28466.271} C_VEL
LIN {X 0,Y 85.551,Z 552.168,A -85,B 0,C 180,E1 -28475.102,E2 -28475.102} C_VEL
LIN {X 0,Y 89.595,Z 553.211,A -85,B 0,C 180,E1 -28478.868,E2 -28478.868} C_VEL
LIN {X 0,Y 82.483,Z 558.303,A -85,B 0,C 180,E1 -28483.592,E2 -28483.592} C_VEL
LIN {X 0,Y 75.88,Z 562.562,A -85,B 0,C 180,E1 -28489.582,E2 -28489.582} C_VEL
LIN {X 0,Y 72.195,Z 564.86,A -85,B 0,C 180,E1 -28494.26,E2 -28494.26} C_VEL
LIN {X 0,Y 69.15,Z 566.707,A -85,B 0,C 180,E1 -28499.456,E2 -28499.456} C_VEL
LIN {X 0,Y 65.329,Z 569.267,A -85,B 0,C 180,E1 -28511.17,E2 -28511.17} C_VEL
LIN {X 0,Y 64.615,Z 570.01,A -85,B 0,C 180,E1 -28518.206,E2 -28518.206} C_VEL
LIN {X 0,Y 64.749,Z 570.248,A -85,B 0,C 180,E1 -28523.767,E2 -28523.767} C_VEL
LIN {X 0,Y 65.374,Z 570.114,A -85,B 0,C 180,E1 -28529.999,E2 -28529.999} C_VEL
LIN {X 0,Y 64.458,Z 568.346,A -85,B 0,C 180,E1 -28541.105,E2 -28541.105} C_VEL
LIN {X 0,Y 65.703,Z 565.319,A -85,B 0,C 180,E1 -28551.985,E2 -28551.985} C_VEL
LIN {X 0,Y 68.655,Z 561.615,A -85,B 0,C 180,E1 -28560.785,E2 -28560.785} C_VEL
LIN {X 0,Y 73.254,Z 556.852,A -85,B 0,C 180,E1 -28568.579,E2 -28568.579} C_VEL
LIN {X 0,Y 77.622,Z 551.744,A -85,B 0,C 180,E1 -28574.707,E2 -28574.707} C_VEL
LIN {X 0,Y 83.189,Z 544.408,A -85,B 0,C 180,E1 -28581.394,E2 -28581.394} C_VEL
LIN {X 0,Y 88.561,Z 536.325,A -85,B 0,C 180,E1 -28586.984,E2 -28586.984} C_VEL
LIN {X 0,Y 93.624,Z 527.473,A -85,B 0,C 180,E1 -28591.887,E2 -28591.887} C_VEL
LIN {X 0,Y 95.682,Z 523.44,A -85,B 0,C 180,E1 -28593.851,E2 -28593.851} C_VEL
LIN {X 0,Y 96.15,Z 522.141,A -85,B 0,C 180,E1 -28594.569,E2 -28594.569} C_VEL
LIN {X 0,Y 96.601,Z 515.878,A -85,B 0,C 180,E1 -28599.825,E2 -28599.825} C_VEL
LIN {X 0,Y 96.641,Z 510.434,A -85,B 0,C 180,E1 -28605.255,E2 -28605.255} C_VEL
LIN {X 0,Y 96.694,Z 506.761,A -85,B 0,C 180,E1 -28609.531,E2 -28609.531} C_VEL
LIN {X 0,Y 96.397,Z 504.281,A -85,B 0,C 180,E1 -28613.722,E2 -28613.722} C_VEL
LIN {X 0,Y 96.279,Z 503.296,A -85,B 0,C 180,E1 -28615.815,E2 -28615.815} C_VEL
LIN {X 0,Y 95.9,Z 502.181,A -85,B 0,C 180,E1 -28620.001,E2 -28620.001} C_VEL
LIN {X 0,Y 95.094,Z 502.506,A -85,B 0,C 180,E1 -28628.501,E2 -28628.501} C_VEL
LIN {X 0,Y 94.742,Z 504.422,A -85,B 0,C 180,E1 -28635.348,E2 -28635.348} C_VEL
LIN {X 0,Y 94.88,Z 506.985,A -85,B 0,C 180,E1 -28641.739,E2 -28641.739} C_VEL
LIN {X 0,Y 95.039,Z 509.453,A -85,B 0,C 180,E1 -28646.34,E2 -28646.34} C_VEL
LIN {X 0,Y 95.128,Z 512.579,A -85,B 0,C 180,E1 -28651.143,E2 -28651.143} C_VEL
LIN {X 0,Y 94.975,Z 516.499,A -85,B 0,C 180,E1 -28656.299,E2 -28656.299} C_VEL
LIN {X 0,Y 94.449,Z 521.194,A -85,B 0,C 180,E1 -28661.919,E2 -28661.919} C_VEL
LIN {X 0,Y 94.141,Z 522.73,A -85,B 0,C 180,E1 -28663.693,E2 -28663.693} C_VEL
LIN {X 0,Y 89.989,Z 527.756,A -85,B 0,C 180,E1 -28666.895,E2 -28666.895} C_VEL
LIN {X 0,Y 84.682,Z 533.483,A -85,B 0,C 180,E1 -28671.506,E2 -28671.506} C_VEL
LIN {X 0,Y 79.009,Z 539.089,A -85,B 0,C 180,E1 -28677.744,E2 -28677.744} C_VEL
LIN {X 0,Y 74.257,Z 543.504,A -85,B 0,C 180,E1 -28684.793,E2 -28684.793} C_VEL
LIN {X 0,Y 70.22,Z 547.092,A -85,B 0,C 180,E1 -28693.255,E2 -28693.255} C_VEL
LIN {X 0,Y 67.378,Z 549.88,A -85,B 0,C 180,E1 -28704.014,E2 -28704.014} C_VEL
LIN {X 0,Y 67.129,Z 551.285,A -85,B 0,C 180,E1 -28716.011,E2 -28716.011} C_VEL
LIN {X 0,Y 67.327,Z 551.339,A -85,B 0,C 180,E1 -28718.658,E2 -28718.658} C_VEL
LIN {X 0,Y 67.103,Z 551.512,A -85,B 0,C 180,E1 -28722.061,E2 -28722.061} C_VEL
LIN {X 0,Y 64.529,Z 551.667,A -85,B 0,C 180,E1 -28733.633,E2 -28733.633} C_VEL
LIN {X 0,Y 65.386,Z 551.249,A -85,B 0,C 180,E1 -28737.031,E2 -28737.031} C_VEL
LIN {X 0,Y 71.322,Z 548.911,A -85,B 0,C 180,E1 -28746.246,E2 -28746.246} C_VEL
LIN {X 0,Y 77.235,Z 545.864,A -85,B 0,C 180,E1 -28753.283,E2 -28753.283} C_VEL
LIN {X 0,Y 83.747,Z 541.931,A -85,B 0,C 180,E1 -28759.052,E2 -28759.052} C_VEL
LIN {X 0,Y 90.989,Z 536.769,A -85,B 0,C 180,E1 -28764.198,E2 -28764.198} C_VEL
LIN {X 0,Y 93.547,Z 534.781,A -85,B 0,C 180,E1 -28765.733,E2 -28765.733} C_VEL
LIN {X 0,Y 94.195,Z 533.294,A -85,B 0,C 180,E1 -28768.514,E2 -28768.514} C_VEL
LIN {X 0,Y 89.53,Z 535.05,A -85,B 0,C 180,E1 -28771.9,E2 -28771.9} C_VEL
LIN {X 0,Y 84.648,Z 537.201,A -85,B 0,C 180,E1 -28775.471,E2 -28775.471} C_VEL
LIN {X 0,Y 71.527,Z 544.226,A -85,B 0,C 180,E1 -28794.36,E2 -28794.36} C_VEL
LIN {X 0,Y 69.788,Z 550.342,A -85,B 0,C 180,E1 -28817.584,E2 -28817.584} C_VEL
LIN {X 0,Y 76.833,Z 554.278,A -85,B 0,C 180,E1 -28833.286,E2 -28833.286} C_VEL
LIN {X 0,Y 80.477,Z 555.461,A -85,B 0,C 180,E1 -28837.683,E2 -28837.683} C_VEL
LIN {X 0,Y 80.424,Z 555.726,A -85,B 0,C 180,E1 -28838.14,E2 -28838.14} C_VEL
LIN {X 0,Y 72.838,Z 560.298,A -85,B 0,C 180,E1 -28843.641,E2 -28843.641} C_VEL
LIN {X 0,Y 66.563,Z 563.884,A -85,B 0,C 180,E1 -28850.689,E2 -28850.689} C_VEL
LIN {X 0,Y 63.115,Z 565.718,A -85,B 0,C 180,E1 -28856.166,E2 -28856.166} C_VEL
LIN {X 0,Y 58.61,Z 568.259,A -85,B 0,C 180,E1 -28868.914,E2 -28868.914} C_VEL
LIN {X 0,Y 57.588,Z 569.021,A -85,B 0,C 180,E1 -28877.5,E2 -28877.5} C_VEL
LIN {X 0,Y 57.668,Z 569.217,A -85,B 0,C 180,E1 -28882.998,E2 -28882.998} C_VEL
LIN {X 0,Y 58.252,Z 569.076,A -85,B 0,C 180,E1 -28889.998,E2 -28889.998} C_VEL
LIN {X 0,Y 57.428,Z 567.416,A -85,B 0,C 180,E1 -28901.757,E2 -28901.757} C_VEL
LIN {X 0,Y 59.088,Z 564.231,A -85,B 0,C 180,E1 -28914.599,E2 -28914.599} C_VEL
LIN {X 0,Y 62.621,Z 560.517,A -85,B 0,C 180,E1 -28924.134,E2 -28924.134} C_VEL
LIN {X 0,Y 67.773,Z 555.725,A -85,B 0,C 180,E1 -28932.378,E2 -28932.378} C_VEL
LIN {X 0,Y 72.368,Z 550.762,A -85,B 0,C 180,E1 -28938.607,E2 -28938.607} C_VEL
LIN {X 0,Y 78.709,Z 543.18,A -85,B 0,C 180,E1 -28945.682,E2 -28945.682} C_VEL
LIN {X 0,Y 84.314,Z 535.503,A -85,B 0,C 180,E1 -28951.065,E2 -28951.065} C_VEL
LIN {X 0,Y 89.659,Z 527.011,A -85,B 0,C 180,E1 -28955.871,E2 -28955.871} C_VEL
LIN {X 0,Y 90.512,Z 525.496,A -85,B 0,C 180,E1 -28956.621,E2 -28956.621} C_VEL
LIN {X 0,Y 90.994,Z 523.807,A -85,B 0,C 180,E1 -28957.944,E2 -28957.944} C_VEL
LIN {X 0,Y 91.722,Z 518.275,A -85,B 0,C 180,E1 -28963.302,E2 -28963.302} C_VEL
LIN {X 0,Y 91.996,Z 515.187,A -85,B 0,C 180,E1 -28966.752,E2 -28966.752} C_VEL
LIN {X 0,Y 92.307,Z 511.352,A -85,B 0,C 180,E1 -28971.799,E2 -28971.799} C_VEL
LIN {X 0,Y 92.232,Z 509.416,A -85,B 0,C 180,E1 -28975.631,E2 -28975.631} C_VEL
LIN {X 0,Y 91.959,Z 508.139,A -85,B 0,C 180,E1 -28980.001,E2 -28980.001} C_VEL
LIN {X 0,Y 91.031,Z 508.348,A -85,B 0,C 180,E1 -28987.195,E2 -28987.195} C_VEL
LIN {X 0,Y 90.946,Z 508.485,A -85,B 0,C 180,E1 -28988.892,E2 -28988.892} C_VEL
LIN {X 0,Y 90.545,Z 509.615,A -85,B 0,C 180,E1 -28993.466,E2 -28993.466} C_VEL
LIN {X 0,Y 90.288,Z 512.22,A -85,B 0,C 180,E1 -29000.922,E2 -29000.922} C_VEL
LIN {X 0,Y 90.158,Z 514.374,A -85,B 0,C 180,E1 -29005.388,E2 -29005.388} C_VEL
LIN {X 0,Y 89.868,Z 517.508,A -85,B 0,C 180,E1 -29010.658,E2 -29010.658} C_VEL
LIN {X 0,Y 89.37,Z 521.051,A -85,B 0,C 180,E1 -29015.837,E2 -29015.837} C_VEL
LIN {X 0,Y 88.508,Z 524.935,A -85,B 0,C 180,E1 -29020.966,E2 -29020.966} C_VEL
LIN {X 0,Y 86.186,Z 527.615,A -85,B 0,C 180,E1 -29022.787,E2 -29022.787} C_VEL
LIN {X 0,Y 79.318,Z 534.609,A -85,B 0,C 180,E1 -29028.354,E2 -29028.354} C_VEL
LIN {X 0,Y 73.173,Z 540.187,A -85,B 0,C 180,E1 -29034.812,E2 -29034.812} C_VEL
LIN {X 0,Y 67.973,Z 544.582,A -85,B 0,C 180,E1 -29042.273,E2 -29042.273} C_VEL
LIN {X 0,Y 63.828,Z 547.946,A -85,B 0,C 180,E1 -29050.713,E2 -29050.713} C_VEL
LIN {X 0,Y 60.395,Z 550.922,A -85,B 0,C 180,E1 -29063.319,E2 -29063.319} C_VEL
LIN {X 0,Y 59.895,Z 551.811,A -85,B 0,C 180,E1 -29070.001,E2 -29070.001} C_VEL
LIN {X 0,Y 60.339,Z 552.345,A -85,B 0,C 180,E1 -29079.217,E2 -29079.217} C_VEL
LIN {X 0,Y 62.336,Z 552.166,A -85,B 0,C 180,E1 -29089.771,E2 -29089.771} C_VEL
LIN {X 0,Y 65.386,Z 551.249,A -85,B 0,C 180,E1 -29097.031,E2 -29097.031} C_VEL
LIN {X 0,Y 67.368,Z 550.446,A -85,B 0,C 180,E1 -29101.772,E2 -29101.772} C_VEL
LIN {X 0,Y 69.797,Z 548.812,A -85,B 0,C 180,E1 -29109.7,E2 -29109.7} C_VEL
LIN {X 0,Y 72.288,Z 547.077,A -85,B 0,C 180,E1 -29115.665,E2 -29115.665} C_VEL
LIN {X 0,Y 75.113,Z 545.335,A -85,B 0,C 180,E1 -29119.506,E2 -29119.506} C_VEL
LIN {X 0,Y 76.296,Z 544.63,A -85,B 0,C 180,E1 -29120.595,E2 -29120.595} C_VEL
LIN {X 0,Y 84.421,Z 539.545,A -85,B 0,C 180,E1 -29126.358,E2 -29126.358} C_VEL
LIN {X 0,Y 85.672,Z 538.695,A -85,B 0,C 180,E1 -29127.135,E2 -29127.135} C_VEL
LIN {X 0,Y 85.573,Z 538.292,A -85,B 0,C 180,E1 -29128.69,E2 -29128.69} C_VEL
LIN {X 0,Y 78.003,Z 541.23,A -85,B 0,C 180,E1 -29134.292,E2 -29134.292} C_VEL
LIN {X 0,Y 65.059,Z 547.579,A -85,B 0,C 180,E1 -29153.798,E2 -29153.798} C_VEL
LIN {X 0,Y 63.583,Z 553.461,A -85,B 0,C 180,E1 -29179.365,E2 -29179.365} C_VEL
LIN {X 0,Y 71.48,Z 557.219,A -85,B 0,C 180,E1 -29196.151,E2 -29196.151} C_VEL
LIN {X 0,Y 70.738,Z 557.93,A -85,B 0,C 180,E1 -29197.36,E2 -29197.36} C_VEL
LIN {X 0,Y 63.396,Z 561.812,A -85,B 0,C 180,E1 -29203.895,E2 -29203.895} C_VEL
LIN {X 0,Y 57.336,Z 564.73,A -85,B 0,C 180,E1 -29212.2,E2 -29212.2} C_VEL
LIN {X 0,Y 52.023,Z 567.253,A -85,B 0,C 180,E1 -29226.089,E2 -29226.089} C_VEL
LIN {X 0,Y 50.597,Z 568.186,A -85,B 0,C 180,E1 -29242.014,E2 -29242.014} C_VEL
LIN {X 0,Y 51.128,Z 568.038,A -85,B 0,C 180,E1 -29249.998,E2 -29249.998} C_VEL
LIN {X 0,Y 50.394,Z 566.496,A -85,B 0,C 180,E1 -29262.523,E2 -29262.523} C_VEL
LIN {X 0,Y 52.642,Z 563.143,A -85,B 0,C 180,E1 -29277.855,E2 -29277.855} C_VEL
LIN {X 0,Y 56.845,Z 559.417,A -85,B 0,C 180,E1 -29288.181,E2 -29288.181} C_VEL
LIN {X 0,Y 62.399,Z 554.797,A -85,B 0,C 180,E1 -29296.533,E2 -29296.533} C_VEL
LIN {X 0,Y 68.906,Z 548.33,A -85,B 0,C 180,E1 -29304.68,E2 -29304.68} C_VEL
LIN {X 0,Y 75.747,Z 540.679,A -85,B 0,C 180,E1 -29311.435,E2 -29311.435} C_VEL
LIN {X 0,Y 82.136,Z 532.44,A -85,B 0,C 180,E1 -29316.899,E2 -29316.899} C_VEL
LIN {X 0,Y 84.77,Z 528.603,A -85,B 0,C 180,E1 -29319.092,E2 -29319.092} C_VEL
LIN {X 0,Y 85.633,Z 527.088,A -85,B 0,C 180,E1 -29320.076,E2 -29320.076} C_VEL
LIN {X 0,Y 86.609,Z 522.721,A -85,B 0,C 180,E1 -29324.709,E2 -29324.709} C_VEL
LIN {X 0,Y 87.177,Z 519.722,A -85,B 0,C 180,E1 -29328.371,E2 -29328.371} C_VEL
LIN {X 0,Y 87.724,Z 516.179,A -85,B 0,C 180,E1 -29333.603,E2 -29333.603} C_VEL
LIN {X 0,Y 87.769,Z 515.32,A -85,B 0,C 180,E1 -29335.408,E2 -29335.408} C_VEL
LIN {X 0,Y 87.657,Z 513.878,A -85,B 0,C 180,E1 -29340.001,E2 -29340.001} C_VEL
LIN {X 0,Y 86.998,Z 513.786,A -85,B 0,C 180,E1 -29344.634,E2 -29344.634} C_VEL
LIN {X 0,Y 86.445,Z 514.267,A -85,B 0,C 180,E1 -29349.359,E2 -29349.359} C_VEL
LIN {X 0,Y 85.858,Z 515.46,A -85,B 0,C 180,E1 -29354.216,E2 -29354.216} C_VEL
LIN {X 0,Y 85.496,Z 516.99,A -85,B 0,C 180,E1 -29359.198,E2 -29359.198} C_VEL
LIN {X 0,Y 85.106,Z 519.128,A -85,B 0,C 180,E1 -29364.388,E2 -29364.388} C_VEL
LIN {X 0,Y 84.425,Z 522.13,A -85,B 0,C 180,E1 -29369.966,E2 -29369.966} C_VEL
LIN {X 0,Y 83.431,Z 525.946,A -85,B 0,C 180,E1 -29376.134,E2 -29376.134} C_VEL
LIN {X 0,Y 83.002,Z 527.176,A -85,B 0,C 180,E1 -29377.977,E2 -29377.977} C_VEL
LIN {X 0,Y 79.062,Z 531.243,A -85,B 0,C 180,E1 -29380.925,E2 -29380.925} C_VEL
LIN {X 0,Y 71.936,Z 537.7,A -85,B 0,C 180,E1 -29386.853,E2 -29386.853} C_VEL
LIN {X 0,Y 65.591,Z 542.848,A -85,B 0,C 180,E1 -29393.893,E2 -29393.893} C_VEL
LIN {X 0,Y 60.245,Z 546.865,A -85,B 0,C 180,E1 -29402.186,E2 -29402.186} C_VEL
LIN {X 0,Y 57.262,Z 549.004,A -85,B 0,C 180,E1 -29408.397,E2 -29408.397} C_VEL
LIN {X 0,Y 53.423,Z 551.964,A -85,B 0,C 180,E1 -29422.442,E2 -29422.442} C_VEL
LIN {X 0,Y 52.867,Z 552.844,A -85,B 0,C 180,E1 -29430.002,E2 -29430.002} C_VEL
LIN {X 0,Y 53.169,Z 553.319,A -85,B 0,C 180,E1 -29437.597,E2 -29437.597} C_VEL
LIN {X 0,Y 55.768,Z 553.166,A -85,B 0,C 180,E1 -29452.216,E2 -29452.216} C_VEL
LIN {X 0,Y 59.14,Z 552.26,A -85,B 0,C 180,E1 -29459.995,E2 -29459.995} C_VEL
LIN {X 0,Y 65.781,Z 549.876,A -85,B 0,C 180,E1 -29469.871,E2 -29469.871} C_VEL
LIN {X 0,Y 72.226,Z 546.836,A -85,B 0,C 180,E1 -29477.066,E2 -29477.066} C_VEL
LIN {X 0,Y 76.296,Z 544.63,A -85,B 0,C 180,E1 -29480.595,E2 -29480.595} C_VEL
LIN {X 0,Y 77.193,Z 543.948,A -85,B 0,C 180,E1 -29482.203,E2 -29482.203} C_VEL
LIN {X 0,Y 76.99,Z 543.572,A -85,B 0,C 180,E1 -29484.715,E2 -29484.715} C_VEL
LIN {X 0,Y 75.343,Z 543.744,A -85,B 0,C 180,E1 -29488.031,E2 -29488.031} C_VEL
LIN {X 0,Y 73.389,Z 544.253,A -85,B 0,C 180,E1 -29490.557,E2 -29490.557} C_VEL
LIN {X 0,Y 67.665,Z 546.202,A -85,B 0,C 180,E1 -29496.833,E2 -29496.833} C_VEL
LIN {X 0,Y 62.454,Z 548.345,A -85,B 0,C 180,E1 -29503.933,E2 -29503.933} C_VEL
LIN {X 0,Y 55.939,Z 553.437,A -85,B 0,C 180,E1 -29527.216,E2 -29527.216} C_VEL
LIN {X 0,Y 59.458,Z 557.423,A -85,B 0,C 180,E1 -29548.216,E2 -29548.216} C_VEL
LIN {X 0,Y 62.496,Z 558.624,A -85,B 0,C 180,E1 -29554.212,E2 -29554.212} C_VEL
LIN {X 0,Y 61.223,Z 559.685,A -85,B 0,C 180,E1 -29556.527,E2 -29556.527} C_VEL
LIN {X 0,Y 56.292,Z 561.93,A -85,B 0,C 180,E1 -29561.486,E2 -29561.486} C_VEL
LIN {X 0,Y 51.894,Z 563.743,A -85,B 0,C 180,E1 -29567.376,E2 -29567.376} C_VEL
LIN {X 0,Y 45.587,Z 566.244,A -85,B 0,C 180,E1 -29582.449,E2 -29582.449} C_VEL
LIN {X 0,Y 43.552,Z 567.156,A -85,B 0,C 180,E1 -29600.712,E2 -29600.712} C_VEL
LIN {X 0,Y 44.002,Z 566.999,A -85,B 0,C 180,E1 -29609.998,E2 -29609.998} C_VEL
LIN {X 0,Y 43.361,Z 565.584,A -85,B 0,C 180,E1 -29623.475,E2 -29623.475} C_VEL
LIN {X 0,Y 46.426,Z 562.055,A -85,B 0,C 180,E1 -29641.992,E2 -29641.992} C_VEL
LIN {X 0,Y 51.416,Z 558.315,A -85,B 0,C 180,E1 -29653.112,E2 -29653.112} C_VEL
LIN {X 0,Y 57.26,Z 553.951,A -85,B 0,C 180,E1 -29661.331,E2 -29661.331} C_VEL
LIN {X 0,Y 64.892,Z 547.136,A -85,B 0,C 180,E1 -29670.044,E2 -29670.044} C_VEL
LIN {X 0,Y 71.635,Z 540.288,A -85,B 0,C 180,E1 -29676.106,E2 -29676.106} C_VEL
LIN {X 0,Y 78.009,Z 532.895,A -85,B 0,C 180,E1 -29681.075,E2 -29681.075} C_VEL
LIN {X 0,Y 80.003,Z 530.313,A -85,B 0,C 180,E1 -29682.6,E2 -29682.6} C_VEL
LIN {X 0,Y 80.595,Z 529.222,A -85,B 0,C 180,E1 -29683.576,E2 -29683.576} C_VEL
LIN {X 0,Y 81.84,Z 525.225,A -85,B 0,C 180,E1 -29688.465,E2 -29688.465} C_VEL
LIN {X 0,Y 82.565,Z 522.422,A -85,B 0,C 180,E1 -29692.665,E2 -29692.665} C_VEL
LIN {X 0,Y 82.96,Z 520.96,A -85,B 0,C 180,E1 -29695.141,E2 -29695.141} C_VEL
LIN {X 0,Y 83.013,Z 519.354,A -85,B 0,C 180,E1 -29700.001,E2 -29700.001} C_VEL
LIN {X 0,Y 82.305,Z 519.254,A -85,B 0,C 180,E1 -29704.899,E2 -29704.899} C_VEL
LIN {X 0,Y 81.613,Z 519.812,A -85,B 0,C 180,E1 -29709.918,E2 -29709.918} C_VEL
LIN {X 0,Y 80.646,Z 521.419,A -85,B 0,C 180,E1 -29716.545,E2 -29716.545} C_VEL
LIN {X 0,Y 80.291,Z 522.595,A -85,B 0,C 180,E1 -29720.496,E2 -29720.496} C_VEL
LIN {X 0,Y 79.397,Z 525.078,A -85,B 0,C 180,E1 -29726.27,E2 -29726.27} C_VEL
LIN {X 0,Y 78.073,Z 528.428,A -85,B 0,C 180,E1 -29732.692,E2 -29732.692} C_VEL
LIN {X 0,Y 77.351,Z 529.921,A -85,B 0,C 180,E1 -29735.144,E2 -29735.144} C_VEL
LIN {X 0,Y 69.473,Z 536.85,A -85,B 0,C 180,E1 -29740.651,E2 -29740.651} C_VEL
LIN {X 0,Y 62.251,Z 542.375,A -85,B 0,C 180,E1 -29747.362,E2 -29747.362} C_VEL
LIN {X 0,Y 55.932,Z 546.735,A -85,B 0,C 180,E1 -29755.569,E2 -29755.569} C_VEL
LIN {X 0,Y 50.811,Z 550.06,A -85,B 0,C 180,E1 -29765.486,E2 -29765.486} C_VEL
LIN {X 0,Y 46.466,Z 553.005,A -85,B 0,C 180,E1 -29781.303,E2 -29781.303} C_VEL
LIN {X 0,Y 45.84,Z 553.877,A -85,B 0,C 180,E1 -29790.002,E2 -29790.002} C_VEL
LIN {X 0,Y 46.21,Z 554.336,A -85,B 0,C 180,E1 -29798.75,E2 -29798.75} C_VEL
LIN {X 0,Y 49.329,Z 554.166,A -85,B 0,C 180,E1 -29815.306,E2 -29815.306} C_VEL
LIN {X 0,Y 52.427,Z 553.479,A -85,B 0,C 180,E1 -29822.428,E2 -29822.428} C_VEL
LIN {X 0,Y 56.267,Z 552.362,A -85,B 0,C 180,E1 -29828.649,E2 -29828.649} C_VEL
LIN {X 0,Y 60.551,Z 550.841,A -85,B 0,C 180,E1 -29834.142,E2 -29834.142} C_VEL
LIN {X 0,Y 67.541,Z 547.825,A -85,B 0,C 180,E1 -29841.365,E2 -29841.365} C_VEL
LIN {X 0,Y 75.262,Z 543.789,A -85,B 0,C 180,E1 -29847.187,E2 -29847.187} C_VEL
LIN {X 0,Y 75.979,Z 543.175,A -85,B 0,C 180,E1 -29848.787,E2 -29848.787} C_VEL
LIN {X 0,Y 62.454,Z 548.345,A -85,B 0,C 180,E1 -29863.933,E2 -29863.933} C_VEL
LIN {X 0,Y 59.433,Z 549.802,A -85,B 0,C 180,E1 -29868.525,E2 -29868.525} C_VEL
LIN {X 0,Y 50.476,Z 554.813,A -85,B 0,C 180,E1 -29883.835,E2 -29883.835} C_VEL
LIN {X 0,Y 49.25,Z 556.174,A -85,B 0,C 180,E1 -29890.26,E2 -29890.26} C_VEL
LIN {X 0,Y 49.24,Z 556.547,A -85,B 0,C 180,E1 -29892.498,E2 -29892.498} C_VEL
LIN {X 0,Y 53.571,Z 559.679,A -85,B 0,C 180,E1 -29911.651,E2 -29911.651} C_VEL
LIN {X 0,Y 51.85,Z 560.952,A -85,B 0,C 180,E1 -29915.58,E2 -29915.58} C_VEL
LIN {X 0,Y 46.905,Z 562.756,A -85,B 0,C 180,E1 -29921.478,E2 -29921.478} C_VEL
LIN {X 0,Y 39.408,Z 565.236,A -85,B 0,C 180,E1 -29937.652,E2 -29937.652} C_VEL
LIN {X 0,Y 36.518,Z 566.122,A -85,B 0,C 180,E1 -29958.902,E2 -29958.902} C_VEL
LIN {X 0,Y 36.855,Z 565.957,A -85,B 0,C 180,E1 -29969.998,E2 -29969.998} C_VEL
LIN {X 0,Y 36.349,Z 564.668,A -85,B 0,C 180,E1 -29984.824,E2 -29984.824} C_VEL
LIN {X 0,Y 39.041,Z 561.979,A -85,B 0,C 180,E1 -30002.685,E2 -30002.685} C_VEL
LIN {X 0,Y 44.261,Z 558.555,A -85,B 0,C 180,E1 -30015.603,E2 -30015.603} C_VEL
LIN {X 0,Y 51.22,Z 554.062,A -85,B 0,C 180,E1 -30025.411,E2 -30025.411} C_VEL
LIN {X 0,Y 58.811,Z 548.204,A -85,B 0,C 180,E1 -30033.668,E2 -30033.668} C_VEL
LIN {X 0,Y 67.075,Z 540.84,A -85,B 0,C 180,E1 -30040.558,E2 -30040.558} C_VEL
LIN {X 0,Y 74.427,Z 533.174,A -85,B 0,C 180,E1 -30045.761,E2 -30045.761} C_VEL
LIN {X 0,Y 75.64,Z 531.444,A -85,B 0,C 180,E1 -30047.29,E2 -30047.29} C_VEL
LIN {X 0,Y 77.058,Z 528.069,A -85,B 0,C 180,E1 -30052.138,E2 -30052.138} C_VEL
LIN {X 0,Y 77.617,Z 526.525,A -85,B 0,C 180,E1 -30054.878,E2 -30054.878} C_VEL
LIN {X 0,Y 78.045,Z 524.597,A -85,B 0,C 180,E1 -30060.001,E2 -30060.001} C_VEL
LIN {X 0,Y 77.294,Z 524.481,A -85,B 0,C 180,E1 -30065.218,E2 -30065.218} C_VEL
LIN {X 0,Y 76.348,Z 525.119,A -85,B 0,C 180,E1 -30070.61,E2 -30070.61} C_VEL
LIN {X 0,Y 75.451,Z 526.328,A -85,B 0,C 180,E1 -30076.228,E2 -30076.228} C_VEL
LIN {X 0,Y 74.456,Z 528.143,A -85,B 0,C 180,E1 -30082.184,E2 -30082.184} C_VEL
LIN {X 0,Y 73.799,Z 529.417,A -85,B 0,C 180,E1 -30085.376,E2 -30085.376} C_VEL
LIN {X 0,Y 72.352,Z 532.011,A -85,B 0,C 180,E1 -30090.975,E2 -30090.975} C_VEL
LIN {X 0,Y 69.271,Z 534.719,A -85,B 0,C 180,E1 -30093.175,E2 -30093.175} C_VEL
LIN {X 0,Y 62.446,Z 539.933,A -85,B 0,C 180,E1 -30098.02,E2 -30098.02} C_VEL
LIN {X 0,Y 54.881,Z 545.04,A -85,B 0,C 180,E1 -30105.228,E2 -30105.228} C_VEL
LIN {X 0,Y 48.277,Z 549.018,A -85,B 0,C 180,E1 -30114.39,E2 -30114.39} C_VEL
LIN {X 0,Y 44.527,Z 551.117,A -85,B 0,C 180,E1 -30121.74,E2 -30121.74} C_VEL
LIN {X 0,Y 39.557,Z 554.044,A -85,B 0,C 180,E1 -30139.768,E2 -30139.768} C_VEL
LIN {X 0,Y 38.812,Z 554.909,A -85,B 0,C 180,E1 -30150.002,E2 -30150.002} C_VEL
LIN {X 0,Y 39.277,Z 555.352,A -85,B 0,C 180,E1 -30160.31,E2 -30160.31} C_VEL
LIN {X 0,Y 43.077,Z 555.166,A -85,B 0,C 180,E1 -30179.307,E2 -30179.307} C_VEL
LIN {X 0,Y 46.645,Z 554.47,A -85,B 0,C 180,E1 -30187.065,E2 -30187.065} C_VEL
LIN {X 0,Y 50.966,Z 553.335,A -85,B 0,C 180,E1 -30193.592,E2 -30193.592} C_VEL
LIN {X 0,Y 55.719,Z 551.807,A -85,B 0,C 180,E1 -30199.186,E2 -30199.186} C_VEL
LIN {X 0,Y 63.373,Z 548.778,A -85,B 0,C 180,E1 -30206.322,E2 -30206.322} C_VEL
LIN {X 0,Y 66.08,Z 547.574,A -85,B 0,C 180,E1 -30208.307,E2 -30208.307} C_VEL
LIN {X 0,Y 64.224,Z 548.064,A -85,B 0,C 180,E1 -30211.099,E2 -30211.099} C_VEL
LIN {X 0,Y 51.638,Z 553.127,A -85,B 0,C 180,E1 -30232.176,E2 -30232.176} C_VEL
LIN {X 0,Y 49.24,Z 556.547,A -85,B 0,C 180,E1 -30252.498,E2 -30252.498} C_VEL
LIN {X 0,Y 48.964,Z 557.472,A -85,B 0,C 180,E1 -30257.188,E2 -30257.188} C_VEL
LIN {X 0,Y 47.925,Z 558.609,A -85,B 0,C 180,E1 -30261.773,E2 -30261.773} C_VEL
LIN {X 0,Y 45.701,Z 560.201,A -85,B 0,C 180,E1 -30267.783,E2 -30267.783} C_VEL
LIN {X 0,Y 42.679,Z 561.651,A -85,B 0,C 180,E1 -30273.676,E2 -30273.676} C_VEL
LIN {X 0,Y 40.847,Z 562.235,A -85,B 0,C 180,E1 -30276.498,E2 -30276.498} C_VEL
LIN {X 0,Y 33.592,Z 564.224,A -85,B 0,C 180,E1 -30291.119,E2 -30291.119} C_VEL
LIN {X 0,Y 29.542,Z 565.089,A -85,B 0,C 180,E1 -30316.235,E2 -30316.235} C_VEL
LIN {X 0,Y 29.693,Z 564.912,A -85,B 0,C 180,E1 -30329.997,E2 -30329.997} C_VEL
LIN {X 0,Y 29.403,Z 563.733,A -85,B 0,C 180,E1 -30347.045,E2 -30347.045} C_VEL
LIN {X 0,Y 33.228,Z 560.897,A -85,B 0,C 180,E1 -30369.382,E2 -30369.382} C_VEL
LIN {X 0,Y 39.571,Z 557.455,A -85,B 0,C 180,E1 -30383.053,E2 -30383.053} C_VEL
LIN {X 0,Y 47.457,Z 552.923,A -85,B 0,C 180,E1 -30392.688,E2 -30392.688} C_VEL
LIN {X 0,Y 55.911,Z 547.021,A -85,B 0,C 180,E1 -30400.515,E2 -30400.515} C_VEL
LIN {X 0,Y 64.939,Z 539.604,A -85,B 0,C 180,E1 -30406.907,E2 -30406.907} C_VEL
LIN {X 0,Y 69.808,Z 535.026,A -85,B 0,C 180,E1 -30409.931,E2 -30409.931} C_VEL
LIN {X 0,Y 70.994,Z 533.369,A -85,B 0,C 180,E1 -30411.859,E2 -30411.859} C_VEL
LIN {X 0,Y 71.808,Z 531.87,A -85,B 0,C 180,E1 -30414.384,E2 -30414.384} C_VEL
LIN {X 0,Y 72.389,Z 530.628,A -85,B 0,C 180,E1 -30417.029,E2 -30417.029} C_VEL
LIN {X 0,Y 72.703,Z 529.641,A -85,B 0,C 180,E1 -30420.001,E2 -30420.001} C_VEL
LIN {X 0,Y 71.936,Z 529.427,A -85,B 0,C 180,E1 -30425.608,E2 -30425.608} C_VEL
LIN {X 0,Y 70.743,Z 530.158,A -85,B 0,C 180,E1 -30431.461,E2 -30431.461} C_VEL
LIN {X 0,Y 69.624,Z 531.4,A -85,B 0,C 180,E1 -30437.628,E2 -30437.628} C_VEL
LIN {X 0,Y 67.957,Z 533.61,A -85,B 0,C 180,E1 -30444.437,E2 -30444.437} C_VEL
LIN {X 0,Y 67.293,Z 534.487,A -85,B 0,C 180,E1 -30446.717,E2 -30446.717} C_VEL
LIN {X 0,Y 65.861,Z 535.729,A -85,B 0,C 180,E1 -30447.974,E2 -30447.974} C_VEL
LIN {X 0,Y 58.389,Z 541.05,A -85,B 0,C 180,E1 -30452.591,E2 -30452.591} C_VEL
LIN {X 0,Y 50.145,Z 546.136,A -85,B 0,C 180,E1 -30459.573,E2 -30459.573} C_VEL
LIN {X 0,Y 42.767,Z 550.095,A -85,B 0,C 180,E1 -30468.906,E2 -30468.906} C_VEL
LIN {X 0,Y 38.493,Z 552.174,A -85,B 0,C 180,E1 -30476.791,E2 -30476.791} C_VEL
LIN {X 0,Y 32.685,Z 555.083,A -85,B 0,C 180,E1 -30497.586,E2 -30497.586} C_VEL
LIN {X 0,Y 31.784,Z 555.94,A -85,B 0,C 180,E1 -30510.003,E2 -30510.003} C_VEL
LIN {X 0,Y 32.386,Z 556.368,A -85,B 0,C 180,E1 -30522.536,E2 -30522.536} C_VEL
LIN {X 0,Y 37.104,Z 556.166,A -85,B 0,C 180,E1 -30544.63,E2 -30544.63} C_VEL
LIN {X 0,Y 41.252,Z 555.46,A -85,B 0,C 180,E1 -30552.961,E2 -30552.961} C_VEL
LIN {X 0,Y 46.129,Z 554.309,A -85,B 0,C 180,E1 -30559.624,E2 -30559.624} C_VEL
LIN {X 0,Y 51.397,Z 552.772,A -85,B 0,C 180,E1 -30565.132,E2 -30565.132} C_VEL
LIN {X 0,Y 56.135,Z 551.115,A -85,B 0,C 180,E1 -30569.946,E2 -30569.946} C_VEL
LIN {X 0,Y 42.913,Z 556.615,A -85,B 0,C 180,E1 -30599.999,E2 -30599.999} C_VEL
LIN {X 0,Y 45.281,Z 560.602,A -85,B 0,C 180,E1 -30629.608,E2 -30629.608} C_VEL
LIN {X 0,Y 44.208,Z 561.266,A -85,B 0,C 180,E1 -30632.357,E2 -30632.357} C_VEL
LIN {X 0,Y 40.847,Z 562.235,A -85,B 0,C 180,E1 -30636.498,E2 -30636.498} C_VEL
LIN {X 0,Y 36.505,Z 563.303,A -85,B 0,C 180,E1 -30642.274,E2 -30642.274} C_VEL
LIN {X 0,Y 29.007,Z 564.109,A -85,B 0,C 180,E1 -30653.608,E2 -30653.608} C_VEL
LIN {X 0,Y 24.128,Z 564.202,A -85,B 0,C 180,E1 -30667.266,E2 -30667.266} C_VEL
LIN {X 0,Y 22.398,Z 564.03,A -85,B 0,C 180,E1 -30681.291,E2 -30681.291} C_VEL
LIN {X 0,Y 22.385,Z 563.907,A -85,B 0,C 180,E1 -30686.354,E2 -30686.354} C_VEL
LIN {X 0,Y 22.537,Z 563.869,A -85,B 0,C 180,E1 -30689.996,E2 -30689.996} C_VEL
LIN {X 0,Y 22.478,Z 562.819,A -85,B 0,C 180,E1 -30710.294,E2 -30710.294} C_VEL
LIN {X 0,Y 28.053,Z 559.816,A -85,B 0,C 180,E1 -30738.723,E2 -30738.723} C_VEL
LIN {X 0,Y 35.722,Z 556.355,A -85,B 0,C 180,E1 -30752.289,E2 -30752.289} C_VEL
LIN {X 0,Y 44.571,Z 551.779,A -85,B 0,C 180,E1 -30761.094,E2 -30761.094} C_VEL
LIN {X 0,Y 53.883,Z 545.835,A -85,B 0,C 180,E1 -30768.015,E2 -30768.015} C_VEL
LIN {X 0,Y 63.676,Z 538.332,A -85,B 0,C 180,E1 -30773.664,E2 -30773.664} C_VEL
LIN {X 0,Y 65.011,Z 537.181,A -85,B 0,C 180,E1 -30774.378,E2 -30774.378} C_VEL
LIN {X 0,Y 65.907,Z 536.235,A -85,B 0,C 180,E1 -30775.414,E2 -30775.414} C_VEL
LIN {X 0,Y 66.482,Z 535.416,A -85,B 0,C 180,E1 -30776.971,E2 -30776.971} C_VEL
LIN {X 0,Y 67.08,Z 534.309,A -85,B 0,C 180,E1 -30780.001,E2 -30780.001} C_VEL
LIN {X 0,Y 66.258,Z 534.072,A -85,B 0,C 180,E1 -30786.09,E2 -30786.09} C_VEL
LIN {X 0,Y 64.794,Z 534.927,A -85,B 0,C 180,E1 -30792.53,E2 -30792.53} C_VEL
LIN {X 0,Y 63.136,Z 536.395,A -85,B 0,C 180,E1 -30799.509,E2 -30799.509} C_VEL
LIN {X 0,Y 61.138,Z 538.069,A -85,B 0,C 180,E1 -30803.131,E2 -30803.131} C_VEL
LIN {X 0,Y 51.897,Z 543.965,A -85,B 0,C 180,E1 -30808.332,E2 -30808.332} C_VEL
LIN {X 0,Y 43.183,Z 548.629,A -85,B 0,C 180,E1 -30815.539,E2 -30815.539} C_VEL
LIN {X 0,Y 35.146,Z 552.256,A -85,B 0,C 180,E1 -30825.586,E2 -30825.586} C_VEL
LIN {X 0,Y 28.762,Z 554.871,A -85,B 0,C 180,E1 -30840.748,E2 -30840.748} C_VEL
LIN {X 0,Y 24.756,Z 556.969,A -85,B 0,C 180,E1 -30870.004,E2 -30870.004} C_VEL
LIN {X 0,Y 25.57,Z 557.385,A -85,B 0,C 180,E1 -30885.957,E2 -30885.957} C_VEL
LIN {X 0,Y 31.572,Z 557.166,A -85,B 0,C 180,E1 -30911.902,E2 -30911.902} C_VEL
LIN {X 0,Y 36.423,Z 556.448,A -85,B 0,C 180,E1 -30920.521,E2 -30920.521} C_VEL
LIN {X 0,Y 41.918,Z 555.283,A -85,B 0,C 180,E1 -30926.966,E2 -30926.966} C_VEL
LIN {X 0,Y 45.199,Z 554.476,A -85,B 0,C 180,E1 -30932.193,E2 -30932.193} C_VEL
LIN {X 0,Y 35.363,Z 559.525,A -85,B 0,C 180,E1 -30971.461,E2 -30971.461} C_VEL
LIN {X 0,Y 36.84,Z 561.02,A -85,B 0,C 180,E1 -30985.322,E2 -30985.322} C_VEL
LIN {X 0,Y 35.422,Z 561.691,A -85,B 0,C 180,E1 -30989.529,E2 -30989.529} C_VEL
LIN {X 0,Y 28.398,Z 563.213,A -85,B 0,C 180,E1 -31002.054,E2 -31002.054} C_VEL
LIN {X 0,Y 22.676,Z 564.057,A -85,B 0,C 180,E1 -31031.941,E2 -31031.941} C_VEL
LIN {X 0,Y 22.385,Z 563.907,A -85,B 0,C 180,E1 -31046.354,E2 -31046.354} C_VEL
LIN {X 0,Y 22.382,Z 563.64,A -85,B 0,C 180,E1 -31056.165,E2 -31056.165} C_VEL
LIN {X 0,Y 21.906,Z 562.775,A -85,B 0,C 180,E1 -31071.108,E2 -31071.108} C_VEL
LIN {X 0,Y 22.333,Z 560.512,A -85,B 0,C 180,E1 -31096.799,E2 -31096.799} C_VEL
LIN {X 0,Y 25.806,Z 558.223,A -85,B 0,C 180,E1 -31113.801,E2 -31113.801} C_VEL
LIN {X 0,Y 28.767,Z 556.95,A -85,B 0,C 180,E1 -31119.097,E2 -31119.097} C_VEL
LIN {X 0,Y 39.474,Z 552.341,A -85,B 0,C 180,E1 -31128.293,E2 -31128.293} C_VEL
LIN {X 0,Y 49.437,Z 546.82,A -85,B 0,C 180,E1 -31134.322,E2 -31134.322} C_VEL
LIN {X 0,Y 59.622,Z 539.9,A -85,B 0,C 180,E1 -31139.111,E2 -31139.111} C_VEL
LIN {X 0,Y 61.057,Z 538.745,A -85,B 0,C 180,E1 -31140.001,E2 -31140.001} C_VEL
LIN {X 0,Y 60.174,Z 538.506,A -85,B 0,C 180,E1 -31146.708,E2 -31146.708} C_VEL
LIN {X 0,Y 58.095,Z 539.58,A -85,B 0,C 180,E1 -31154.585,E2 -31154.585} C_VEL
LIN {X 0,Y 57.432,Z 540.049,A -85,B 0,C 180,E1 -31156.895,E2 -31156.895} C_VEL
LIN {X 0,Y 55.451,Z 541.316,A -85,B 0,C 180,E1 -31158.096,E2 -31158.096} C_VEL
LIN {X 0,Y 45.764,Z 546.75,A -85,B 0,C 180,E1 -31162.87,E2 -31162.87} C_VEL
LIN {X 0,Y 36.419,Z 551.041,A -85,B 0,C 180,E1 -31169.732,E2 -31169.732} C_VEL
LIN {X 0,Y 27.835,Z 554.29,A -85,B 0,C 180,E1 -31180.765,E2 -31180.765} C_VEL
LIN {X 0,Y 19.231,Z 557.161,A -85,B 0,C 180,E1 -31208.569,E2 -31208.569} C_VEL
LIN {X 0,Y 17.728,Z 557.997,A -85,B 0,C 180,E1 -31230.005,E2 -31230.005} C_VEL
LIN {X 0,Y 18.91,Z 558.401,A -85,B 0,C 180,E1 -31251.822,E2 -31251.822} C_VEL
LIN {X 0,Y 26.753,Z 558.166,A -85,B 0,C 180,E1 -31282.013,E2 -31282.013} C_VEL
LIN {X 0,Y 33.815,Z 557.178,A -85,B 0,C 180,E1 -31291.627,E2 -31291.627} C_VEL
LIN {X 0,Y 35.013,Z 557.015,A -85,B 0,C 180,E1 -31294.518,E2 -31294.518} C_VEL
LIN {X 0,Y 28.707,Z 561.118,A -85,B 0,C 180,E1 -31338.668,E2 -31338.668} C_VEL
LIN {X 0,Y 26.844,Z 561.765,A -85,B 0,C 180,E1 -31345.014,E2 -31345.014} C_VEL
LIN {X 0,Y 19.239,Z 562.799,A -85,B 0,C 180,E1 -31363.056,E2 -31363.056} C_VEL
LIN {X 0,Y 16.052,Z 563.027,A -85,B 0,C 180,E1 -31384.028,E2 -31384.028} C_VEL
LIN {X 0,Y 15.39,Z 562.827,A -85,B 0,C 180,E1 -31409.994,E2 -31409.994} C_VEL
LIN {X 0,Y 15.713,Z 561.896,A -85,B 0,C 180,E1 -31436.562,E2 -31436.562} C_VEL
LIN {X 0,Y 23.941,Z 558.737,A -85,B 0,C 180,E1 -31471.717,E2 -31471.717} C_VEL
LIN {X 0,Y 28.767,Z 556.95,A -85,B 0,C 180,E1 -31479.097,E2 -31479.097} C_VEL
LIN {X 0,Y 33.291,Z 554.979,A -85,B 0,C 180,E1 -31485.102,E2 -31485.102} C_VEL
LIN {X 0,Y 37.47,Z 552.761,A -85,B 0,C 180,E1 -31490.956,E2 -31490.956} C_VEL
LIN {X 0,Y 45.952,Z 547.683,A -85,B 0,C 180,E1 -31500.452,E2 -31500.452} C_VEL
LIN {X 0,Y 50.617,Z 544.822,A -85,B 0,C 180,E1 -31503.407,E2 -31503.407} C_VEL
LIN {X 0,Y 52.25,Z 543.804,A -85,B 0,C 180,E1 -31504.056,E2 -31504.056} C_VEL
LIN {X 0,Y 54.363,Z 542.463,A -85,B 0,C 180,E1 -31505.07,E2 -31505.07} C_VEL
LIN {X 0,Y 52.682,Z 543.022,A -85,B 0,C 180,E1 -31511.054,E2 -31511.054} C_VEL
LIN {X 0,Y 43.523,Z 547.845,A -85,B 0,C 180,E1 -31514.339,E2 -31514.339} C_VEL
LIN {X 0,Y 33.498,Z 552.118,A -85,B 0,C 180,E1 -31519.25,E2 -31519.25} C_VEL
LIN {X 0,Y 23.853,Z 555.348,A -85,B 0,C 180,E1 -31527.889,E2 -31527.889} C_VEL
LIN {X 0,Y 12.959,Z 558.201,A -85,B 0,C 180,E1 -31557.165,E2 -31557.165} C_VEL
LIN {X 0,Y 10.7,Z 559.024,A -85,B 0,C 180,E1 -31590.008,E2 -31590.008} C_VEL
LIN {X 0,Y 12.658,Z 559.418,A -85,B 0,C 180,E1 -31623.736,E2 -31623.736} C_VEL
LIN {X 0,Y 23.1,Z 559.166,A -85,B 0,C 180,E1 -31655.896,E2 -31655.896} C_VEL
LIN {X 0,Y 24.515,Z 559.149,A -85,B 0,C 180,E1 -31660.381,E2 -31660.381} C_VEL
LIN {X 0,Y 21.289,Z 560.926,A -85,B 0,C 180,E1 -31687.923,E2 -31687.923} C_VEL
LIN {X 0,Y 19.988,Z 561.359,A -85,B 0,C 180,E1 -31694.753,E2 -31694.753} C_VEL
LIN {X 0,Y 10.123,Z 561.993,A -85,B 0,C 180,E1 -31726.017,E2 -31726.017} C_VEL
LIN {X 0,Y 8.239,Z 561.785,A -85,B 0,C 180,E1 -31769.989,E2 -31769.989} C_VEL
LIN {X 0,Y 9.822,Z 560.832,A -85,B 0,C 180,E1 -31815.675,E2 -31815.675} C_VEL
LIN {X 0,Y 21.488,Z 557.654,A -85,B 0,C 180,E1 -31848.858,E2 -31848.858} C_VEL
LIN {X 0,Y 31.706,Z 554.157,A -85,B 0,C 180,E1 -31855.903,E2 -31855.903} C_VEL
LIN {X 0,Y 41.097,Z 550.013,A -85,B 0,C 180,E1 -31860.002,E2 -31860.002} C_VEL
LIN {X 0,Y 52.25,Z 543.804,A -85,B 0,C 180,E1 -31864.056,E2 -31864.056} C_VEL
LIN {X 0,Y 51.52,Z 544.141,A -85,B 0,C 180,E1 -31865.013,E2 -31865.013} C_VEL
LIN {X 0,Y 49.628,Z 545.155,A -85,B 0,C 180,E1 -31865.805,E2 -31865.805} C_VEL
LIN {X 0,Y 41.846,Z 549.01,A -85,B 0,C 180,E1 -31867.12,E2 -31867.12} C_VEL
LIN {X 0,Y 30.915,Z 553.534,A -85,B 0,C 180,E1 -31867.67,E2 -31867.67} C_VEL
LIN {X 0,Y 19.684,Z 557.041,A -85,B 0,C 180,E1 -31867.66,E2 -31867.66} C_VEL
LIN {X 0,Y 12.049,Z 558.782,A -85,B 0,C 180,E1 -31866.116,E2 -31866.116} C_VEL
LIN {X 0,Y 1.088,Z 560.742,A -85,B 0,C 180,E1 -31769.919,E2 -31769.919} C_VEL
LIN {X 0,Y 7.819,Z 560.955,A -85,B 0,C 180,E1 -31679.992,E2 -31679.992} C_VEL
LIN {X 0,Y 14.102,Z 560.754,A -85,B 0,C 180,E1 -31675.432,E2 -31675.432} C_VEL
LIN {X 0,Y 14.38,Z 560.481,A -85,B 0,C 180,E1 -31667.839,E2 -31667.839} C_VEL
LIN {X 0,Y 7.851,Z 560.434,A -85,B 0,C 180,E1 -31653.552,E2 -31653.552} C_VEL
LIN {X 0,Y 3.671,Z 560.049,A -85,B 0,C 180,E1 -31590.024,E2 -31590.024} C_VEL
LIN {X 0,Y 8.023,Z 559.241,A -85,B 0,C 180,E1 -31528.867,E2 -31528.867} C_VEL
LIN {X 0,Y 21.485,Z 556.405,A -85,B 0,C 180,E1 -31511.107,E2 -31511.107} C_VEL
LIN {X 0,Y 21.299,Z 556.572,A -85,B 0,C 180,E1 -31508.185,E2 -31508.185} C_VEL
LIN {X 0,Y 12.049,Z 558.782,A -85,B 0,C 180,E1 -31506.116,E2 -31506.116} C_VEL
LIN {X 0,Y 10.44,Z 560.745,A -85,B 0,C 180,E1 -31505.327,E2 -31505.327} C_VEL
LIN {X 0,Y 10.44,Z 600,A -85,B 0,C 180,E1 -31505.327,E2 -31505.327} C_VEL
LIN {X 0,Y 10.44,Z 600,A -85,B 0,C 180,E1 -31505.327,E2 -31505.327}

QRS_NEXT_CUT()

QRS_NEXT()
QRS_HOME()

END
